{attribute 'reflection'}
FUNCTION_BLOCK FB_RS485_EASTRON_SDM630_MQTT EXTENDS FB_MQTT_BASE IMPLEMENTS I_RS485_DEVICE
  VAR
    {attribute 'noinit'}
    {attribute 'instance-path'}
    sInstancePath : STRING(GVL_MQTT.MQTT_TOPIC_LEN);  (* object's full instance name *)
    bIsDataUpdated : BOOL := FALSE;
    fbTimerData : TON;
    stStep : ST_RS485_STEP;  (* One read covers the whole measurement block: function 4 (input registers), 64 words from 16#000C (phase 1 power) to 16#004B (total export energy). Reading it in one stStep keeps the values consistent with each other and costs the bus one slot instead of 26. Filled by FB_init in code rather than by a declaration initialiser, which a script cannot revise once the compiler has stored it. *)
    fbMqttDiscoveryDevice : FB_EASTRON_SDM_MQTT_DISCOVERY_DEVICE;  (* Owned rather than referenced, unlike the 1-Wire sensors which share a gateway device from the GVL: a meter is one Home Assistant device on its own, so there is nothing to share and self-wiring has nothing to look up. *)
  END_VAR
  VAR_OUTPUT
    L1_ACTIVEPOWER : REAL := 0;
    L2_ACTIVEPOWER : REAL := 0;  (* L1 Active Power. SDM630 input register 16#000C. *)
    L3_ACTIVEPOWER : REAL := 0;  (* L2 Active Power. SDM630 input register 16#000E. *)
    L1_VA : REAL := 0;  (* L3 Active Power. SDM630 input register 16#0010. *)
    L2_VA : REAL := 0;  (* L1 Apparent Power. SDM630 input register 16#0012. *)
    L3_VA : REAL := 0;  (* L2 Apparent Power. SDM630 input register 16#0014. *)
    L1_VAR : REAL := 0;  (* L3 Apparent Power. SDM630 input register 16#0016. *)
    L2_VAR : REAL := 0;  (* L1 Reactive Power. SDM630 input register 16#0018. *)
    L3_VAR : REAL := 0;  (* L2 Reactive Power. SDM630 input register 16#001A. *)
    L1_PF : REAL := 0;  (* L3 Reactive Power. SDM630 input register 16#001C. *)
    L2_PF : REAL := 0;  (* L1 Power Factor. SDM630 input register 16#001E. *)
    L3_PF : REAL := 0;  (* L2 Power Factor. SDM630 input register 16#0020. *)
    L1_PHI : REAL := 0;  (* L3 Power Factor. SDM630 input register 16#0022. *)
    L2_PHI : REAL := 0;  (* L1 Phase Angle. SDM630 input register 16#0024. *)
    L3_PHI : REAL := 0;  (* L2 Phase Angle. SDM630 input register 16#0026. *)
    AVG_LN_V : REAL := 0;  (* L3 Phase Angle. SDM630 input register 16#0028. *)
    AVG_LINE_I : REAL := 0;  (* Average L-iN Voltage. SDM630 input register 16#002A. *)
    SUM_LINE_I : REAL := 0;  (* Average Line Current. SDM630 input register 16#002C. *)
    ACTIVEPOWER : REAL := 0;  (* Sum of Line Currents. SDM630 input register 16#002E. *)
    TOTAL_VA : REAL := 0;  (* Active Power. SDM630 input register 16#0034. *)
    TOTAL_VAR : REAL := 0;  (* Total Apparent Power. SDM630 input register 16#0038. *)
    TOTAL_PF : REAL := 0;  (* Total Reactive Power. SDM630 input register 16#003C. *)
    TOTAL_PHI : REAL := 0;  (* Total Power Factor. SDM630 input register 16#003E. *)
    FREQUENCY : REAL := 0;  (* Total Phase Angle. SDM630 input register 16#0042. *)
    TOTAL_IMPORT_ENERGY : REAL := 0;  (* Frequency. SDM630 input register 16#0046. *)
    TOTAL_EXPORT_ENERGY : REAL := 0;  (* Total Import Energy. SDM630 input register 16#0048. *)
    DataAvailable : BOOL := FALSE;  (* Total Export Energy. SDM630 input register 16#004A. *)
    Error : BOOL := FALSE;
  END_VAR

            (* --- self-wiring prologue ----------------------------------------------------
   Makes the InitMqtt and InitMqttDiscovery calls optional. Set FriendlyName at
   the declaration site and this block wires itself from GVL_MQTT on its
   first cyclic call, then announces itself to Home Assistant.

   Deliberately in the body rather than in FB_init: it dereferences GVL members
   and reads the reflection instance path, and doing that during initialisation
   would rely on an ordering nothing enforces and the compiler cannot check. The
   body is the same lifecycle phase the init actions used, so this is not merely
   safe, it is the phase that already works today.

   The wiring calls this block's own unmodified InitMqtt / InitMqttDiscovery
   methods, so anything published - topics and discovery JSON alike - is produced
   by exactly the code that produces it today. Only the trigger moved.

   Dormant while FriendlyName is empty, so existing projects and existing call
   sites keep working untouched.

   A block wired this way MUST be called cyclically. An instance whose body never
   runs is now unwired and absent from Home Assistant, where the init action used
   to wire it regardless. Nothing warns about that.  *)
IF FriendlyName <> '' THEN

	IF NOT bInitMqttDone THEN
		THIS^.InitMqtt(
			MQTTPublishPrefix := ADR(GVL_MQTT.MqttPubRS485Prefix),
			pMqttPublishQueue := ADR(GVL_MQTT.fbMqttPublishQueue));
	END_IF

	IF bInitMqttDone AND NOT bInitMqttDiscoveryDone THEN
		THIS^.InitMqttDiscovery(
			Device := ADR(THIS^.fbMqttDiscoveryDevice),
			DeviceName := FriendlyName);
	END_IF

END_IF

fbTimerData();

(* Publish on change of data rather than on a timer: ProcessDataArray sets the
   flag when a response arrives, so the publish rate follows DataPollingInterval
   and nothing is republished while the bus is quiet. PubMqttMessage is a no-op
   until InitMqtt has run, so this needs no further guard. *)
IF bIsDataUpdated THEN
	bIsDataUpdated := FALSE;

	PubMqttMessage(Suffix := '/L1_ACTP', Data := REAL_TO_STRING(L1_ACTIVEPOWER));
	PubMqttMessage(Suffix := '/L2_ACTP', Data := REAL_TO_STRING(L2_ACTIVEPOWER));
	PubMqttMessage(Suffix := '/L3_ACTP', Data := REAL_TO_STRING(L3_ACTIVEPOWER));
	PubMqttMessage(Suffix := '/L1_VA', Data := REAL_TO_STRING(L1_VA));
	PubMqttMessage(Suffix := '/L2_VA', Data := REAL_TO_STRING(L2_VA));
	PubMqttMessage(Suffix := '/L3_VA', Data := REAL_TO_STRING(L3_VA));
	PubMqttMessage(Suffix := '/L1_VAR', Data := REAL_TO_STRING(L1_VAR));
	PubMqttMessage(Suffix := '/L2_VAR', Data := REAL_TO_STRING(L2_VAR));
	PubMqttMessage(Suffix := '/L3_VAR', Data := REAL_TO_STRING(L3_VAR));
	PubMqttMessage(Suffix := '/L1_PF', Data := REAL_TO_STRING(L1_PF));
	PubMqttMessage(Suffix := '/L2_PF', Data := REAL_TO_STRING(L2_PF));
	PubMqttMessage(Suffix := '/L3_PF', Data := REAL_TO_STRING(L3_PF));
	PubMqttMessage(Suffix := '/L1_PHI', Data := REAL_TO_STRING(L1_PHI));
	PubMqttMessage(Suffix := '/L2_PHI', Data := REAL_TO_STRING(L2_PHI));
	PubMqttMessage(Suffix := '/L3_PHI', Data := REAL_TO_STRING(L3_PHI));
	PubMqttMessage(Suffix := '/AVG_V', Data := REAL_TO_STRING(AVG_LN_V));
	PubMqttMessage(Suffix := '/AVG_I', Data := REAL_TO_STRING(AVG_LINE_I));
	PubMqttMessage(Suffix := '/SUM_I', Data := REAL_TO_STRING(SUM_LINE_I));
	PubMqttMessage(Suffix := '/ACTP', Data := REAL_TO_STRING(ACTIVEPOWER));
	PubMqttMessage(Suffix := '/TOT_VA', Data := REAL_TO_STRING(TOTAL_VA));
	PubMqttMessage(Suffix := '/TOT_VAR', Data := REAL_TO_STRING(TOTAL_VAR));
	PubMqttMessage(Suffix := '/TOT_PF', Data := REAL_TO_STRING(TOTAL_PF));
	PubMqttMessage(Suffix := '/TOT_PHI', Data := REAL_TO_STRING(TOTAL_PHI));
	PubMqttMessage(Suffix := '/FREQ', Data := REAL_TO_STRING(FREQUENCY));
	PubMqttMessage(Suffix := '/IMPE', Data := REAL_TO_STRING(TOTAL_IMPORT_ENERGY));
	PubMqttMessage(Suffix := '/EXPE', Data := REAL_TO_STRING(TOTAL_EXPORT_ENERGY));
END_IF
          

METHOD HasWork : E_RS485_WORK_LEVEL
                  IF fbTimerData.Q THEN
	HasWork := E_RS485_WORK_LEVEL.POLL;
ELSE
	HasWork := E_RS485_WORK_LEVEL.NONE;
END_IF

                
END_METHOD

METHOD OnStepResult
  VAR_INPUT
    StepIndex : INT;
    Failed : BOOL;
    pData : POINTER TO A_RS485_READ_BUFFER;
    Count : INT;
  END_VAR
                  THIS^.Error := Failed;
THIS^.fbTimerData.IN := TRUE;

IF NOT Failed AND Count >= 64 THEN
	(* Every value is a big-endian IEEE float across two consecutive words, so the
	   word index is the register offset from 16#000C doubled. Gaps below are
	   registers the SDM630 reserves. *)
	THIS^.L1_ACTIVEPOWER := F_SWAP_WORDS_TO_REAL(pData^[0], pData^[1]);	// 16#000C L1 Active Power
	THIS^.L2_ACTIVEPOWER := F_SWAP_WORDS_TO_REAL(pData^[2], pData^[3]);	// 16#000E L2 Active Power
	THIS^.L3_ACTIVEPOWER := F_SWAP_WORDS_TO_REAL(pData^[4], pData^[5]);	// 16#0010 L3 Active Power
	THIS^.L1_VA := F_SWAP_WORDS_TO_REAL(pData^[6], pData^[7]);	// 16#0012 L1 Apparent Power
	THIS^.L2_VA := F_SWAP_WORDS_TO_REAL(pData^[8], pData^[9]);	// 16#0014 L2 Apparent Power
	THIS^.L3_VA := F_SWAP_WORDS_TO_REAL(pData^[10], pData^[11]);	// 16#0016 L3 Apparent Power
	THIS^.L1_VAR := F_SWAP_WORDS_TO_REAL(pData^[12], pData^[13]);	// 16#0018 L1 Reactive Power
	THIS^.L2_VAR := F_SWAP_WORDS_TO_REAL(pData^[14], pData^[15]);	// 16#001A L2 Reactive Power
	THIS^.L3_VAR := F_SWAP_WORDS_TO_REAL(pData^[16], pData^[17]);	// 16#001C L3 Reactive Power
	THIS^.L1_PF := F_SWAP_WORDS_TO_REAL(pData^[18], pData^[19]);	// 16#001E L1 Power Factor
	THIS^.L2_PF := F_SWAP_WORDS_TO_REAL(pData^[20], pData^[21]);	// 16#0020 L2 Power Factor
	THIS^.L3_PF := F_SWAP_WORDS_TO_REAL(pData^[22], pData^[23]);	// 16#0022 L3 Power Factor
	THIS^.L1_PHI := F_SWAP_WORDS_TO_REAL(pData^[24], pData^[25]);	// 16#0024 L1 Phase Angle
	THIS^.L2_PHI := F_SWAP_WORDS_TO_REAL(pData^[26], pData^[27]);	// 16#0026 L2 Phase Angle
	THIS^.L3_PHI := F_SWAP_WORDS_TO_REAL(pData^[28], pData^[29]);	// 16#0028 L3 Phase Angle
	THIS^.AVG_LN_V := F_SWAP_WORDS_TO_REAL(pData^[30], pData^[31]);	// 16#002A Average L-iN Voltage
	THIS^.AVG_LINE_I := F_SWAP_WORDS_TO_REAL(pData^[32], pData^[33]);	// 16#002C Average Line Current
	THIS^.SUM_LINE_I := F_SWAP_WORDS_TO_REAL(pData^[34], pData^[35]);	// 16#002E Sum of Line Currents
	THIS^.ACTIVEPOWER := F_SWAP_WORDS_TO_REAL(pData^[40], pData^[41]);	// 16#0034 Active Power
	THIS^.TOTAL_VA := F_SWAP_WORDS_TO_REAL(pData^[44], pData^[45]);	// 16#0038 Total Apparent Power
	THIS^.TOTAL_VAR := F_SWAP_WORDS_TO_REAL(pData^[48], pData^[49]);	// 16#003C Total Reactive Power
	THIS^.TOTAL_PF := F_SWAP_WORDS_TO_REAL(pData^[50], pData^[51]);	// 16#003E Total Power Factor
	THIS^.TOTAL_PHI := F_SWAP_WORDS_TO_REAL(pData^[54], pData^[55]);	// 16#0042 Total Phase Angle
	THIS^.FREQUENCY := F_SWAP_WORDS_TO_REAL(pData^[58], pData^[59]);	// 16#0046 Frequency
	THIS^.TOTAL_IMPORT_ENERGY := F_SWAP_WORDS_TO_REAL(pData^[60], pData^[61]);	// 16#0048 Total Import Energy
	THIS^.TOTAL_EXPORT_ENERGY := F_SWAP_WORDS_TO_REAL(pData^[62], pData^[63]);	// 16#004A Total Export Energy

	THIS^.DataAvailable := TRUE;
	THIS^.bIsDataUpdated := TRUE;
END_IF

                
END_METHOD

METHOD BuildTransaction : INT
  VAR_INPUT
    pSteps : POINTER TO A_RS485_STEP_LIST;
  END_VAR
  VAR
    iN : INT;
  END_VAR
                  IF fbTimerData.Q THEN
	pSteps^[0]			:= stStep;
	fbTimerData.IN		:= FALSE;
	BuildTransaction	:= 1;
ELSE
	BuildTransaction := 0;
END_IF

                
END_METHOD

METHOD InitMqttDiscovery
  VAR_INPUT
    Device : POINTER TO FB_EASTRON_SDM_MQTT_DISCOVERY_DEVICE;
    DeviceName : STRING(50);
    Model : STRING(20) := 'SDM630';
    overruleId : STRING(255) := '';
  END_VAR
  VAR
    id : STRING(255);
  END_VAR
                  (* Announces the meter as a device of its own, then one sensor entity per
   measurement. StateClass is what puts the two kWh totals into the Home
   Assistant energy dashboard; the instantaneous values are 'measurement' and
   power factor, phase angle, voltage, current and frequency carry none. *)
IF bInitMqttDone AND NOT bInitMqttDiscoveryDone THEN

	id := SUPER^.ResolveEntityId(overruleId := overruleId);

	Device^.initEastronDevice(
		name := DeviceName,
		id := id,
		Model := Model,
		availabilityTopic1 := GVL_MQTT.MqttAvailabilityTopic,
		availabilityTopic2 := CONCAT(THIS^.sMQTTPublishTopic, '/availability'),
		availabilityOnline := GVL_MQTT.MqttAvailabilityOnlinePayload,
		availabilityOffline := GVL_MQTT.MqttAvailabilityOfflinePayload,
		MqttDiscoveryPrefix := GVL_MQTT.MqttHADiscoveryPrefix,
		MqttDiagnosticTopic := CONCAT(THIS^.sMQTTPublishTopic, '/diagnostic'),
		pMqttPublishQueue := ADR(GVL_MQTT.fbMqttPublishQueue));

(* This device publishes from the RS485 task, so its messages take that
   task's queue lane. A lane may only ever have one producing task. *)
Device^.SetLane(Lane := GVL_MQTT.MQTT_LANE_RS485);

	Device^.CreateSensorEntity(
		Name := 'L1 Active Power',
		Id := CONCAT(id, '_L1_ACTP'),
		StateTopic := CONCAT(THIS^.sMQTTPublishTopic, '/L1_ACTP'),
		DeviceClass := 'power',
		StateClass := 'measurement',
		UnitOfMeasurement := 'W');

	Device^.CreateSensorEntity(
		Name := 'L2 Active Power',
		Id := CONCAT(id, '_L2_ACTP'),
		StateTopic := CONCAT(THIS^.sMQTTPublishTopic, '/L2_ACTP'),
		DeviceClass := 'power',
		StateClass := 'measurement',
		UnitOfMeasurement := 'W');

	Device^.CreateSensorEntity(
		Name := 'L3 Active Power',
		Id := CONCAT(id, '_L3_ACTP'),
		StateTopic := CONCAT(THIS^.sMQTTPublishTopic, '/L3_ACTP'),
		DeviceClass := 'power',
		StateClass := 'measurement',
		UnitOfMeasurement := 'W');

	Device^.CreateSensorEntity(
		Name := 'L1 Apparent Power',
		Id := CONCAT(id, '_L1_VA'),
		StateTopic := CONCAT(THIS^.sMQTTPublishTopic, '/L1_VA'),
		DeviceClass := 'apparent_power',
		StateClass := 'measurement',
		UnitOfMeasurement := 'VA');

	Device^.CreateSensorEntity(
		Name := 'L2 Apparent Power',
		Id := CONCAT(id, '_L2_VA'),
		StateTopic := CONCAT(THIS^.sMQTTPublishTopic, '/L2_VA'),
		DeviceClass := 'apparent_power',
		StateClass := 'measurement',
		UnitOfMeasurement := 'VA');

	Device^.CreateSensorEntity(
		Name := 'L3 Apparent Power',
		Id := CONCAT(id, '_L3_VA'),
		StateTopic := CONCAT(THIS^.sMQTTPublishTopic, '/L3_VA'),
		DeviceClass := 'apparent_power',
		StateClass := 'measurement',
		UnitOfMeasurement := 'VA');

	Device^.CreateSensorEntity(
		Name := 'L1 Reactive Power',
		Id := CONCAT(id, '_L1_VAR'),
		StateTopic := CONCAT(THIS^.sMQTTPublishTopic, '/L1_VAR'),
		DeviceClass := 'reactive_power',
		StateClass := 'measurement',
		UnitOfMeasurement := 'var');

	Device^.CreateSensorEntity(
		Name := 'L2 Reactive Power',
		Id := CONCAT(id, '_L2_VAR'),
		StateTopic := CONCAT(THIS^.sMQTTPublishTopic, '/L2_VAR'),
		DeviceClass := 'reactive_power',
		StateClass := 'measurement',
		UnitOfMeasurement := 'var');

	Device^.CreateSensorEntity(
		Name := 'L3 Reactive Power',
		Id := CONCAT(id, '_L3_VAR'),
		StateTopic := CONCAT(THIS^.sMQTTPublishTopic, '/L3_VAR'),
		DeviceClass := 'reactive_power',
		StateClass := 'measurement',
		UnitOfMeasurement := 'var');

	Device^.CreateSensorEntity(
		Name := 'L1 Power Factor',
		Id := CONCAT(id, '_L1_PF'),
		StateTopic := CONCAT(THIS^.sMQTTPublishTopic, '/L1_PF'),
		DeviceClass := 'power_factor',
		UnitOfMeasurement := '');

	Device^.CreateSensorEntity(
		Name := 'L2 Power Factor',
		Id := CONCAT(id, '_L2_PF'),
		StateTopic := CONCAT(THIS^.sMQTTPublishTopic, '/L2_PF'),
		DeviceClass := 'power_factor',
		UnitOfMeasurement := '');

	Device^.CreateSensorEntity(
		Name := 'L3 Power Factor',
		Id := CONCAT(id, '_L3_PF'),
		StateTopic := CONCAT(THIS^.sMQTTPublishTopic, '/L3_PF'),
		DeviceClass := 'power_factor',
		UnitOfMeasurement := '');

	Device^.CreateSensorEntity(
		Name := 'L1 Phase Angle',
		Id := CONCAT(id, '_L1_PHI'),
		StateTopic := CONCAT(THIS^.sMQTTPublishTopic, '/L1_PHI'),
		DeviceClass := '',
		UnitOfMeasurement := '°');

	Device^.CreateSensorEntity(
		Name := 'L2 Phase Angle',
		Id := CONCAT(id, '_L2_PHI'),
		StateTopic := CONCAT(THIS^.sMQTTPublishTopic, '/L2_PHI'),
		DeviceClass := '',
		UnitOfMeasurement := '°');

	Device^.CreateSensorEntity(
		Name := 'L3 Phase Angle',
		Id := CONCAT(id, '_L3_PHI'),
		StateTopic := CONCAT(THIS^.sMQTTPublishTopic, '/L3_PHI'),
		DeviceClass := '',
		UnitOfMeasurement := '°');

	Device^.CreateSensorEntity(
		Name := 'Average L-N Voltage',
		Id := CONCAT(id, '_AVG_V'),
		StateTopic := CONCAT(THIS^.sMQTTPublishTopic, '/AVG_V'),
		DeviceClass := 'voltage',
		UnitOfMeasurement := 'V');

	Device^.CreateSensorEntity(
		Name := 'Average Line Current',
		Id := CONCAT(id, '_AVG_I'),
		StateTopic := CONCAT(THIS^.sMQTTPublishTopic, '/AVG_I'),
		DeviceClass := 'current',
		UnitOfMeasurement := 'A');

	Device^.CreateSensorEntity(
		Name := 'Sum of Line Currents',
		Id := CONCAT(id, '_SUM_I'),
		StateTopic := CONCAT(THIS^.sMQTTPublishTopic, '/SUM_I'),
		DeviceClass := 'current',
		UnitOfMeasurement := 'A');

	Device^.CreateSensorEntity(
		Name := 'Active Power',
		Id := CONCAT(id, '_ACTP'),
		StateTopic := CONCAT(THIS^.sMQTTPublishTopic, '/ACTP'),
		DeviceClass := 'power',
		StateClass := 'measurement',
		UnitOfMeasurement := 'W');

	Device^.CreateSensorEntity(
		Name := 'Total Apparent Power',
		Id := CONCAT(id, '_TOT_VA'),
		StateTopic := CONCAT(THIS^.sMQTTPublishTopic, '/TOT_VA'),
		DeviceClass := 'apparent_power',
		StateClass := 'measurement',
		UnitOfMeasurement := 'VA');

	Device^.CreateSensorEntity(
		Name := 'Total Reactive Power',
		Id := CONCAT(id, '_TOT_VAR'),
		StateTopic := CONCAT(THIS^.sMQTTPublishTopic, '/TOT_VAR'),
		DeviceClass := 'reactive_power',
		StateClass := 'measurement',
		UnitOfMeasurement := 'var');

	Device^.CreateSensorEntity(
		Name := 'Total Power Factor',
		Id := CONCAT(id, '_TOT_PF'),
		StateTopic := CONCAT(THIS^.sMQTTPublishTopic, '/TOT_PF'),
		DeviceClass := 'power_factor',
		UnitOfMeasurement := '');

	Device^.CreateSensorEntity(
		Name := 'Total Phase Angle',
		Id := CONCAT(id, '_TOT_PHI'),
		StateTopic := CONCAT(THIS^.sMQTTPublishTopic, '/TOT_PHI'),
		DeviceClass := '',
		UnitOfMeasurement := '°');

	Device^.CreateSensorEntity(
		Name := 'Frequency',
		Id := CONCAT(id, '_FREQ'),
		StateTopic := CONCAT(THIS^.sMQTTPublishTopic, '/FREQ'),
		DeviceClass := 'frequency',
		UnitOfMeasurement := 'Hz');

	Device^.CreateSensorEntity(
		Name := 'Total Import Energy',
		Id := CONCAT(id, '_IMP_ENERG'),
		StateTopic := CONCAT(THIS^.sMQTTPublishTopic, '/IMPE'),
		DeviceClass := 'energy',
		StateClass := 'total_increasing',
		UnitOfMeasurement := 'kWh');

	Device^.CreateSensorEntity(
		Name := 'Total Export Energy',
		Id := CONCAT(id, '_EXP_ENERG'),
		StateTopic := CONCAT(THIS^.sMQTTPublishTopic, '/EXPE'),
		DeviceClass := 'energy',
		StateClass := 'total_increasing',
		UnitOfMeasurement := 'kWh');

	bInitMqttDiscoveryDone := TRUE;
END_IF
                
END_METHOD

METHOD PubMqttMessage
  VAR_INPUT
    Suffix : STRING(100);
    Data : STRING(100);
  END_VAR
                  IF bInitMqttDone THEN
		pMqttPublishQueue^.AddMessageOn(Lane := GVL_MQTT.MQTT_LANE_RS485,
			Payload := Data,
			Topic := CONCAT(THIS^.sMQTTPublishTopic, Suffix),
			Qos := MQTT.QoS.ExactlyOnce,
			MqttRetain := FALSE
		);
END_IF
                
END_METHOD

METHOD InitMqtt
  VAR_INPUT
    MQTTPublishPrefix : POINTER TO STRING;
    pMqttPublishQueue : POINTER TO FB_MQTT_PUBLISH_QUEUE;
  END_VAR
                  SUPER^._sInstancePath := THIS^.sInstancePath; // Due to reflection its location is important

(*pass trough*)
THIS^.pMqttPublishQueue := pMqttPublishQueue;
THIS^.psMqttPublishTopicPrefix := MQTTPublishPrefix;

SUPER^.InitBaseMqtt();
                
END_METHOD

METHOD FB_init : BOOL
  VAR_INPUT
    bInitRetains : BOOL;  (* TRUE: the retain variables are initialized (reset warm / reset cold) *)
    bInCopyCode : BOOL;  (* TRUE: the instance will be copied to the copy code afterward (online change) *)
    DeviceAddress : BYTE;  (* Modbus slave address of the meter. *)
    DataPollingInterval : TIME;  (* How often the meter is read. One read covers all 26 measurements. *)
  END_VAR
                  (* Modbus address and poll rate describe the wiring, not a mode, so they are
   fixed for the life of the instance and belong here rather than in a runtime
   setter. Note the consequence: changing either afterwards means editing the
   declaration in the IDE - CODESYS stores an instance's FB_init arguments beside
   the declaration text, where no script can reach them. *)
THIS^.stStep.DeviceId		:= DeviceAddress;
THIS^.stStep.FunctionCode	:= 4;
THIS^.stStep.Address		:= 12;	(* 16#000C, phase 1 active power *)
THIS^.stStep.Quantity		:= 64;	(* through 16#004B, total export energy *)

THIS^.fbTimerData.PT := DataPollingInterval;
THIS^.fbTimerData.IN := TRUE;

FB_init := TRUE;

                
END_METHOD

METHOD OnTransactionDone
  VAR_INPUT
    StepsRun : INT;
    Failures : INT;
  END_VAR
                  (* One announcement per transaction, at the point the bus is released. *)
IF StepsRun > 0 AND Failures >= StepsRun THEN
	PubMqttMessage(Suffix := '/availability', Data := 'offline');
ELSIF StepsRun > 0 THEN
	PubMqttMessage(Suffix := '/availability', Data := 'online');
END_IF

                
END_METHOD

(* Nothing to commission on this device. See I_RS485_DEVICE.GetCommissioning. *)
METHOD GetCommissioning : BOOL
  VAR_INPUT
    BusBaudrate : UDINT;
    pRequest : POINTER TO ST_RS485_COMMISSION_REQUEST;
  END_VAR
                  (* Nothing to commission. This device is configured on the device itself - switches,
   a display, or a factory setting that already matches this bus - so it answers at
   whatever the bus runs at and there is nothing for the commissioner to write.

   Which is the ordinary case: the cost of the whole mechanism, for a device like
   this one, is this method call once at startup. *)
GetCommissioning := FALSE;

                
END_METHOD
END_FUNCTION_BLOCK

{attribute 'reflection'}
FUNCTION_BLOCK FB_RS485_ESERA_OWD_MQTT EXTENDS FB_MQTT_BASE IMPLEMENTS I_RS485_DEVICE
  VAR
    {attribute 'noinit'}
    {attribute 'instance-path'}
    sInstancePath : STRING(GVL_MQTT.MQTT_TOPIC_LEN);  (* object's full instance name *)
    OwdNumber : UINT;
    fbTimerData : TON;
    stStep : ST_RS485_STEP;  (* One read of the gateway's per-sensor block: function 3, 17 holding registers from OwdNumber * 100. Filled by FB_init in code. *)
    pMqttDiscoveryDevice : POINTER TO FB_1WIRE_MQTT_DISCOVERY_DEVICE;
    uiAllowedErrorCount : UINT := 3;
    uiCurrentErrorCount : UINT := 0;
  END_VAR
  VAR_OUTPUT
    OWD_VOLTAGE : REAL := 0;
    TEMPERATURE : REAL := 0;
    HUMIDITY : REAL := 0;
    DEW_POINT : REAL := 0;
    AIR_QUALITY : REAL := 0;
    BRIGHTNESS : REAL := 0;
    DataAvailable : BOOL := FALSE;
    Error : BOOL := FALSE;
  END_VAR

            fbTimerData();


          

METHOD HasWork : E_RS485_WORK_LEVEL
                  IF fbTimerData.Q THEN
	HasWork := E_RS485_WORK_LEVEL.POLL;
ELSE
	HasWork := E_RS485_WORK_LEVEL.NONE;
END_IF

                
END_METHOD

METHOD OnStepResult
  VAR_INPUT
    StepIndex : INT;
    Failed : BOOL;
    pData : POINTER TO A_RS485_READ_BUFFER;
    Count : INT;
  END_VAR
                  THIS^.fbTimerData.IN := TRUE;

(* Register 12 is the gateway's own status word for this sensor: non-zero means
   the gateway answered but the 1-Wire device behind it did not. A short reply
   is treated the same way - there is no status to trust. *)
IF Failed OR Count < 17 OR WORD_TO_INT(pData^[12]) <> 0 THEN
	THIS^.Error := TRUE;
	(* A single miss is normal on a 1-Wire bus, so availability only drops after
	   uiAllowedErrorCount of them in a row. *)
	IF THIS^.uiCurrentErrorCount >= THIS^.uiAllowedErrorCount THEN
		PubMqttMessage(Suffix := '/availability', Data := 'offline');
	END_IF
	THIS^.uiCurrentErrorCount := THIS^.uiCurrentErrorCount + 1;
	RETURN;
END_IF

THIS^.Error := FALSE;
THIS^.DataAvailable := TRUE;
THIS^.uiCurrentErrorCount := 0;
PubMqttMessage(Suffix := '/availability', Data := 'online');

IF bInitMqttDiscoveryDone THEN
	THIS^.pMqttDiscoveryDevice^.SendDeviceUpdate(Model := WORD_TO_STRING(pData^[16]));
END_IF

// Data handling
IF pData^[16] = 11151 OR pData^[16] = 11152 THEN // Temperature, humidity & air quality
	ProcessTemperature(pData^[0]);
	ProcessOwdVoltage(pData^[2]);
	ProcessHumidity(pData^[4]);
	ProcessDewPoint(pData^[6]);
	ProcessAirQuality(pData^[8]);
ELSIF pData^[16] = 11102 OR pData^[16] = 11113 OR pData^[16] = 11120 OR pData^[16] = 11148 OR pData^[16] = 11150 OR pData^[16] = 11160 THEN // Temperature, humidity
	ProcessTemperature(pData^[0]);
	ProcessOwdVoltage(pData^[2]);
	ProcessHumidity(pData^[4]);
	ProcessDewPoint(pData^[6]);
ELSIF pData^[16] = 11121 OR pData^[16] = 11132 OR pData^[16] = 11134 OR pData^[16] = 11135 THEN // Temperature, humidity, brightness
	ProcessTemperature(pData^[0]);
	ProcessOwdVoltage(pData^[2]);
	ProcessHumidity(pData^[4]);
	ProcessDewPoint(pData^[6]);
	ProcessBrigthness(pData^[8]);
ELSIF pData^[16] = 1820 THEN // Temperature DS18B20
	ProcessTemperature(pData^[0]);
END_IF

                
END_METHOD

METHOD BuildTransaction : INT
  VAR_INPUT
    pSteps : POINTER TO A_RS485_STEP_LIST;
  END_VAR
  VAR
    iN : INT;
  END_VAR
                  IF fbTimerData.Q THEN
	pSteps^[0]			:= stStep;
	fbTimerData.IN		:= FALSE;
	BuildTransaction	:= 1;
ELSE
	BuildTransaction := 0;
END_IF

                
END_METHOD

METHOD InitMqttDiscovery
  VAR_INPUT
    Device : POINTER TO FB_1WIRE_MQTT_DISCOVERY_DEVICE;
    ParentDevice : POINTER TO FB_PLC_MQTT_DISCOVERY_DEVICE;
    DeviceName : STRING(50);
    SupportsTemperature : BOOL := FALSE;
    SupportsHumidity : BOOL := FALSE;
    SupportsCO2 : BOOL := FALSE;
    SupportsDewPoint : BOOL := FALSE;
    SupportsBrightness : BOOL := FALSE;
    SupportsOwdVoltage : BOOL := FALSE;
  END_VAR
  VAR
    id : STRING(255);
  END_VAR
                  IF bInitMqttDone AND NOT bInitMqttDiscoveryDone THEN
	
	THIS^.pMqttDiscoveryDevice := Device;
	
	id := SUPER^.ResolveEntityId(overruleId := '');
	
	Device^.init1WireDevice(
		name := DeviceName,
		id := id,
		deviceAvailabilityTopic := CONCAT(THIS^.sMQTTPublishTopic, '/availability'),
		deviceDiagnosticTopic := CONCAT(THIS^.sMQTTPublishTopic, '/diagnostic'));

(* This device publishes from the RS485 task, so its messages take that
   task's queue lane. A lane may only ever have one producing task. *)
Device^.SetLane(Lane := GVL_MQTT.MQTT_LANE_RS485);
		
	IF SupportsTemperature THEN
		Device^.CreateSensorEntity(
			Name := 'Temperature',
			Id := CONCAT(id, '_TEMP'),
			StateTopic := CONCAT(THIS^.sMQTTPublishTopic, '/TEMP'),
			DeviceClass := 'temperature',
			UnitOfMeasurement := '°C'); 
	END_IF;	
	
	IF SupportsHumidity THEN
		Device^.CreateSensorEntity(
			Name := 'Humidity',
			Id := CONCAT(id, '_HUM'),
			StateTopic := CONCAT(THIS^.sMQTTPublishTopic, '/HUM'),
			DeviceClass := 'humidity',
			UnitOfMeasurement := '%');
	END_IF;
	
	IF SupportsCO2 THEN
		Device^.CreateSensorEntity(
			Name := 'Carbon Dioxide',
			Id := CONCAT(id, '_CO2'),
			StateTopic := CONCAT(THIS^.sMQTTPublishTopic, '/CO2'),
			DeviceClass := 'carbon_dioxide',
			UnitOfMeasurement := 'ppm');
	END_IF;
	
	IF SupportsDewPoint THEN
		Device^.CreateSensorEntity(
			Name := 'Dew Point',
			Id := CONCAT(id, '_DEWP'),
			StateTopic := CONCAT(THIS^.sMQTTPublishTopic, '/DEWP'),
			DeviceClass := 'temperature',
			UnitOfMeasurement := '°C'); 
	END_IF;	
	
	IF SupportsBrightness THEN
		Device^.CreateSensorEntity(
			Name := 'Brightness',
			Id := CONCAT(id, '_ILLUM'),
			StateTopic := CONCAT(THIS^.sMQTTPublishTopic, '/ILLUM'),
			DeviceClass := 'illuminance');
	END_IF;	
	
	IF SupportsOwdVoltage THEN
		Device^.CreateDiagnosticSensorEntity(
			Name := 'Operating Voltage',
			Id := CONCAT(id, '_OWDV'),
			StateTopic := CONCAT(THIS^.sMQTTPublishTopic, '/OWDV'));
	END_IF;

	bInitMqttDiscoveryDone := TRUE;
END_IF
                
END_METHOD

METHOD InitMqtt
  VAR_INPUT
    MQTTPublishPrefix : POINTER TO STRING;
    pMqttPublishQueue : POINTER TO FB_MQTT_PUBLISH_QUEUE;
  END_VAR
                  SUPER^._sInstancePath := THIS^.sInstancePath; // Due to reflection its location is important

(*pass trough*)
THIS^.pMqttPublishQueue := pMqttPublishQueue;
THIS^.psMqttPublishTopicPrefix:=MQTTPublishPrefix;
SUPER^.InitBaseMqtt();

                
END_METHOD

METHOD PubMqttMessage
  VAR_INPUT
    Suffix : STRING(100);
    Data : STRING(100);
  END_VAR
                  IF bInitMqttDone THEN
		pMqttPublishQueue^.AddMessageOn(Lane := GVL_MQTT.MQTT_LANE_RS485,
			Payload := Data,
			Topic := CONCAT(CONCAT(psMqttPublishTopicPrefix^, MqttPublishTopicSuffix), Suffix),
			Qos := MQTT.QoS.ExactlyOnce,
			MqttRetain := FALSE
		);
END_IF
                
END_METHOD

METHOD ProcessTemperature
  VAR_INPUT
    Data : WORD;
  END_VAR
                  (* Signed: the gateway scales by 100 and encodes two's complement, and both
   of these read below zero on an outdoor sensor. Unsigned turned -1 degree
   into +655.35 and nothing could report frost. *)
THIS^.TEMPERATURE := INT_TO_REAL(WORD_TO_INT(Data)) / 100;
PubMqttMessage(Suffix := '/TEMP', Data := REAL_TO_STRING(TEMPERATURE));
                
END_METHOD

METHOD ProcessOwdVoltage
  VAR_INPUT
    Data : WORD;
  END_VAR
                  THIS^.OWD_VOLTAGE := WORD_TO_REAL(Data);
PubMqttMessage(Suffix := '/OWDV', Data := REAL_TO_STRING(OWD_VOLTAGE));
                
END_METHOD

METHOD ProcessHumidity
  VAR_INPUT
    Data : WORD;
  END_VAR
                  THIS^.HUMIDITY := WORD_TO_REAL(Data) / 100;
PubMqttMessage(Suffix := '/HUM', Data := REAL_TO_STRING(HUMIDITY));
                
END_METHOD

METHOD ProcessDewPoint
  VAR_INPUT
    Data : WORD;
  END_VAR
                  (* Signed: the gateway scales by 100 and encodes two's complement, and both
   of these read below zero on an outdoor sensor. Unsigned turned -1 degree
   into +655.35 and nothing could report frost. *)
THIS^.DEW_POINT := INT_TO_REAL(WORD_TO_INT(Data)) / 100;
PubMqttMessage(Suffix := '/DEWP', Data := REAL_TO_STRING(DEW_POINT));
                
END_METHOD

METHOD ProcessAirQuality
  VAR_INPUT
    Data : WORD;
  END_VAR
                  THIS^.AIR_QUALITY := WORD_TO_REAL(Data) / 100;
PubMqttMessage(Suffix := '/CO2', Data := REAL_TO_STRING(AIR_QUALITY));
                
END_METHOD

METHOD ProcessBrigthness
  VAR_INPUT
    Data : WORD;
  END_VAR
                  THIS^.BRIGHTNESS := WORD_TO_REAL(Data) / 100;
(* /ILLUM, matching the entity id and the StateTopic in InitMqttDiscovery.
   This published to /BNESS, so the illuminance entity never received a value. *)
PubMqttMessage(Suffix := '/ILLUM', Data := REAL_TO_STRING(BRIGHTNESS));
                
END_METHOD

(* FB_Init is always available implicitly and it is used primarily for initialization. The return value is not evaluated. For a specific influence, you can also declare the methods explicitly and provide additional code there with the standard initialization code. You can evaluate the return value. *)
METHOD FB_init : BOOL
  VAR_INPUT
    bInitRetains : BOOL;  (* TRUE: the retain variables are initialized (reset warm / reset cold) *)
    bInCopyCode : BOOL;  (* TRUE: the instance will be copied to the copy code afterward (online change) *)
    DeviceAddress : BYTE;
    OwdNumber : UINT;
    DataPollingInterval : TIME;
  END_VAR
                  THIS^.stStep.DeviceId		:= DeviceAddress;
THIS^.stStep.FunctionCode	:= 3;
THIS^.stStep.Address		:= OwdNumber * 100;
THIS^.stStep.Quantity		:= 17;

THIS^.fbTimerData.PT := DataPollingInterval;
THIS^.OwdNumber := OwdNumber;

THIS^.fbTimerData.IN := TRUE;

FB_Init := TRUE;

                
END_METHOD

METHOD OnTransactionDone
  VAR_INPUT
    StepsRun : INT;
    Failures : INT;
  END_VAR
                  (* Availability for this block is decided in OnStepResult, where the gateway's
   own status register and the consecutive-error count are both in scope. There
   is nothing left to announce here, and announcing it twice would undo the
   error tolerance. *)
;

                
END_METHOD

(* Nothing to commission on this device. See I_RS485_DEVICE.GetCommissioning. *)
METHOD GetCommissioning : BOOL
  VAR_INPUT
    BusBaudrate : UDINT;
    pRequest : POINTER TO ST_RS485_COMMISSION_REQUEST;
  END_VAR
                  (* Nothing to commission. This device is configured on the device itself - switches,
   a display, or a factory setting that already matches this bus - so it answers at
   whatever the bus runs at and there is nothing for the commissioner to write.

   Which is the ordinary case: the cost of the whole mechanism, for a device like
   this one, is this method call once at startup. *)
GetCommissioning := FALSE;

                
END_METHOD
END_FUNCTION_BLOCK

(* Modbus RTU master for the PFC's onboard serial port, behind I_RS485_TRANSPORT. This is the code that was proven on the bench in #182, lifted out of the RS485_RUN action into a block of its own and taught the write function codes it was missing. Two things about this hardware are baked in and deliberate: - Every reply arrives wrapped in glitch bytes - one 00 as the slave's driver enables, another as it releases, because the pair is undriven between frames. Measured across 34 consecutive captures: 34 leading nulls, 34 trailing nulls, 34 wCrc-bDataValid frames once trimmed. So the frame is trimmed and the wCrc judges what is left, rather than the iFirst byte being trusted. - The frame is delimited by silence, which is what RTU actually specifies, not by a byte count read out of the header. The counters are outputs on purpose. They are the only view of line quality this project has without a scope, and LeadNulls climbing in stStep with Ok is the normal healthy picture here, not a fault. *)
FUNCTION_BLOCK FB_RS485_TRANSPORT_RTU IMPLEMENTS I_RS485_TRANSPORT
  VAR_OUTPUT
    PortOpen : BOOL;  (* The serial port is open and usable *)
    PortError : BOOL;  (* SysComOpen2 failed; Reopen to try again *)
    Ok : UDINT;  (* Reply accepted *)
    CrcFail : UDINT;  (* Bytes arrived, wCrc over the trimmed frame was not zero *)
    NoReply : UDINT;  (* Nothing at all before the reply timeout *)
    ShortFrame : UDINT;  (* Too few bytes to be any bDataValid reply *)
    BadAddress : UDINT;  (* A well-formed frame from the wrong slave *)
    BadFunction : UDINT;  (* Right slave, function code we did not ask for *)
    BadEcho : UDINT;  (* Write acknowledged with the wrong address or value *)
    Exceptions : UDINT;  (* Slave answered with an exception reply *)
    LastException : BYTE;  (* Exception code from the most recent one *)
    LeadNulls : UDINT;  (* Not faults. On this hardware both should track Ok almost exactly. *)
    TrailNulls : UDINT;
    LastFailLen : UDINT;  (* The bytes of the most recent frame that would not check out, and how many there were. A counter can say a reply did not frame; only the bytes can say whether it was half a reply, two replies, an echo of the request, or noise - and those want different fixes. *)
    LastFailAddr : BYTE;
    LastFailFunc : BYTE;
    LastFailBytes : STRING(120);
  END_VAR
  VAR
    bConfigured : BOOL;  (* --- port ------------------------------------------------------------ *)
    stSettings : SysCom.SysComSettings;
    hPort : RTS_IEC_HANDLE;
    eRtsResult : RTS_IEC_RESULT;
    bReopenRequest : BOOL;
    GapTime : TIME := TIME#50ms;  (* Line quiet for this long ends a frame *)
    ReplyTimeout : TIME := TIME#1s0ms;  (* Nothing at all by now means no reply *)
    iState : INT;  (* 0 idle, 1 collecting, 2 judging *)
    eOutcome : E_RS485_STEP_STATE := E_RS485_STEP_STATE.IDLE;
    stStep : ST_RS485_STEP;  (* private copy: the caller's scratch is reused *)
    Data : A_RS485_READ_BUFFER;
    iRegCount : INT;
    abyTx : ARRAY[0..31] OF BYTE;  (* 9 + 2*8 for the largest FC16 *)
    iTxLen : INT;  (* payload before the wCrc *)
    abyRx : ARRAY[0..287] OF BYTE;
    udiRxCount : UDINT;
    abyFlush : ARRAY[0..287] OF BYTE;
    fbGap : TON;
    fbReplyTimer : TON;
    bRestartGap : BOOL;
    bRestartReply : BOOL;
    udiN : UDINT;  (* --- scratch ---------------------------------------------------------- *)
    pbyRx : POINTER TO BYTE;
    count : INT;
    iFirst : INT;
    iLast : INT;
    iFrameLen : INT;
    iK : INT;
    wCrc : WORD;
    uiEchoAddr : UINT;
    uiEchoValue : UINT;
    bDataValid : BOOL;
    stConfiguredSettings : SysCom.SysComSettings;  (* What Init bConfigured, saved so RestoreTuning can undo a commissioning sweep without the caller having to remember what it passed in. A sweep changes stSettings in place - that is the only way to reach the port - so the original has to live somewhere or it is gone. *)
    tConfiguredReplyTimeout : TIME;
    tConfiguredGapTime : TIME;
  END_VAR

            
          

METHOD ReadBuffer : POINTER TO A_RS485_READ_BUFFER
                  ReadBuffer := ADR(Data);

                
END_METHOD

METHOD Service : E_RS485_STEP_STATE
                  (* ---------------------------------------------------------------- the port *)
IF bReopenRequest THEN
	bReopenRequest := FALSE;
	IF PortOpen THEN
		SysCom.SysComClose(hPort);
	END_IF
	PortOpen	:= FALSE;
	PortError	:= FALSE;
	iState		:= 0;
	eOutcome		:= E_RS485_STEP_STATE.IDLE;
END_IF

IF bConfigured AND NOT PortOpen AND NOT PortError THEN
	hPort		:= SysCom.SysComOpen2(pSettings := ADR(stSettings), pSettingsEx := 0, pResult := ADR(eRtsResult));
	PortError	:= (hPort = RTS_INVALID_HANDLE OR eRtsResult <> 0);
	PortOpen	:= NOT PortError;
END_IF

(* Both timers are called unconditionally. A TON left with IN true while the
   iState machine is elsewhere goes on counting, and would then fire instantly
   on the next stStep. *)
fbGap(IN := (iState = 1) AND NOT bRestartGap, PT := GapTime);
fbReplyTimer(IN := (iState = 1) AND NOT bRestartReply, PT := ReplyTimeout);
bRestartGap		:= FALSE;
bRestartReply	:= FALSE;

(* ------------------------------------------------------- the stStep in flight *)
CASE iState OF

0:	(* Idle. OK and FAILED were each returned for exactly one cycle, by the
	   return at the bottom of the cycle that reached iState 2. *)
	eOutcome := E_RS485_STEP_STATE.IDLE;

1:	(* Collect until the line has been quiet for GapTime, which is how RTU
	   delimits a frame, or until the slave has clearly not answered at all. *)
	IF udiRxCount < SIZEOF(abyRx) THEN
		pbyRx := ADR(abyRx);
		pbyRx := pbyRx + udiRxCount;
		udiN := SysCom.SysComRead(hPort, pbyRx, SIZEOF(abyRx) - udiRxCount, 0, ADR(eRtsResult));
		IF udiN > 0 THEN
			udiRxCount		:= udiRxCount + udiN;
			bRestartGap	:= TRUE;
		END_IF
	END_IF

	(* A frame whose wCrc already checks out is complete by definition, so there
	   is nothing left to wait for. Waiting anyway costs about three task cycles
	   per stStep, and on a 200 ms task that is most of what a Modbus exchange
	   takes: measured at 1.87 s per stStep before this check, against roughly
	   100 ms of actual wire time at 9600 baud.

	   The silence timer stays as the fallback for everything that does not
	   frame cleanly - a partial reply, a burst of noise, a slave that answers
	   with something we cannot parse. *)
	count := UDINT_TO_INT(udiRxCount);
	IF count >= 5 AND THIS^.Frame() THEN
		iState := 2;
	ELSIF (udiRxCount > 0 AND fbGap.Q) OR fbReplyTimer.Q OR udiRxCount >= SIZEOF(abyRx) THEN
		iState := 2;
	END_IF

2:	THIS^.Judge();
	iState := 0;

END_CASE

Service := eOutcome;

                
END_METHOD

METHOD Start : BOOL
  VAR_INPUT
    pStep : POINTER TO ST_RS485_STEP;
  END_VAR
  VAR
    iI : INT;
    iQty : INT;
  END_VAR
                  Start := FALSE;

IF pStep = 0 OR NOT PortOpen OR iState <> 0 THEN
	RETURN;
END_IF

(* Private copy. The scheduler's stStep list is scratch that it reuses for the
   next device, so nothing may be read back out of it later - the echo checks
   below run against this copy. *)
stStep := pStep^;
iQty := UINT_TO_INT(stStep.Quantity);

CASE stStep.FunctionCode OF

3, 4:	(* read holding / read input registers *)
	IF iQty < 1 OR iQty > (DINT_TO_INT(UPPER_BOUND(Data, 1)) + 1) THEN
		RETURN;
	END_IF
	abyTx[0] := stStep.DeviceId;
	abyTx[1] := stStep.FunctionCode;
	abyTx[2] := UINT_TO_BYTE(SHR(stStep.Address, 8));
	abyTx[3] := UINT_TO_BYTE(stStep.Address AND 16#00FF);
	abyTx[4] := UINT_TO_BYTE(SHR(stStep.Quantity, 8));
	abyTx[5] := UINT_TO_BYTE(stStep.Quantity AND 16#00FF);
	iTxLen := 6;

6:	(* write single register: the value goes where the quantity would *)
	abyTx[0] := stStep.DeviceId;
	abyTx[1] := 16#06;
	abyTx[2] := UINT_TO_BYTE(SHR(stStep.Address, 8));
	abyTx[3] := UINT_TO_BYTE(stStep.Address AND 16#00FF);
	abyTx[4] := WORD_TO_BYTE(SHR(stStep.Data[0], 8));
	abyTx[5] := WORD_TO_BYTE(stStep.Data[0] AND 16#00FF);
	iTxLen := 6;

16:	(* write multiple registers: header, byte count, then the payload *)
	IF iQty < 1 OR iQty > (DINT_TO_INT(UPPER_BOUND(stStep.Data, 1)) + 1) THEN
		RETURN;
	END_IF
	abyTx[0] := stStep.DeviceId;
	abyTx[1] := 16#10;
	abyTx[2] := UINT_TO_BYTE(SHR(stStep.Address, 8));
	abyTx[3] := UINT_TO_BYTE(stStep.Address AND 16#00FF);
	abyTx[4] := UINT_TO_BYTE(SHR(stStep.Quantity, 8));
	abyTx[5] := UINT_TO_BYTE(stStep.Quantity AND 16#00FF);
	abyTx[6] := INT_TO_BYTE(iQty * 2);
	FOR iI := 0 TO iQty - 1 DO
		abyTx[7 + 2 * iI] := WORD_TO_BYTE(SHR(stStep.Data[iI], 8));
		abyTx[8 + 2 * iI] := WORD_TO_BYTE(stStep.Data[iI] AND 16#00FF);
	END_FOR
	iTxLen := 7 + 2 * iQty;

ELSE
	(* Refused, not guessed at. Guessing is precisely the bug this replaces:
	   every function code used to be framed from the read fields, so an FC6
	   write went out as "write register 0 := 0" and its echoed reply was then
	   parsed as though byte 2 were a length. *)
	RETURN;

END_CASE

(* Anything still in the receive buffer belongs to the previous exchange and
   would otherwise be collected as this one's reply. *)
udiN := SysCom.SysComRead(hPort, ADR(abyFlush), SIZEOF(abyFlush), 0, ADR(eRtsResult));

wCrc := THIS^.Crc16(pBuf := ADR(abyTx), Len := iTxLen);
abyTx[iTxLen]		:= WORD_TO_BYTE(wCrc AND 16#00FF);
abyTx[iTxLen + 1]	:= WORD_TO_BYTE(SHR(wCrc, 8));

SysCom.SysComWrite(hPort, ADR(abyTx), INT_TO_UDINT(iTxLen + 2), 100, ADR(eRtsResult));

udiRxCount			:= 0;
iRegCount		:= 0;
bRestartGap		:= TRUE;
bRestartReply	:= TRUE;
eOutcome			:= E_RS485_STEP_STATE.BUSY;
iState			:= 1;
Start			:= TRUE;

                
END_METHOD

METHOD Judge
  VAR
    iBytecount : INT;
    iI : INT;
    bGotFrame : BOOL;
  END_VAR
                  count		:= UDINT_TO_INT(udiRxCount);
bGotFrame	:= THIS^.Frame();

(* Leading glitch bytes are the slave's driver enabling onto an undriven pair,
   trailing ones its releasing. Both are normal on this hardware. *)
IF iFirst > 0 THEN
	LeadNulls := LeadNulls + 1;
END_IF
IF bGotFrame AND iLast < count THEN
	TrailNulls := TrailNulls + 1;
END_IF

iFrameLen	:= iLast - iFirst;
iRegCount	:= 0;
bDataValid		:= FALSE;

IF count = 0 OR (count - iFirst) = 0 THEN
	NoReply := NoReply + 1;

ELSIF (count - iFirst) < 5 THEN
	ShortFrame := ShortFrame + 1;

ELSIF NOT bGotFrame THEN
	CrcFail := CrcFail + 1;

	(* Capture what actually arrived. Two theories about these failures have now
	   been wrong - leading glitch bytes, then a framer that could not
	   resynchronise - and both were argued from counters rather than from
	   bytes. A counter says a frame did not check out; it cannot say whether
	   what arrived was half a reply, two replies, an echo, or noise. Decimal
	   rather than hex because there is no hex helper in scope and the point is
	   to read it off an MQTT topic, not to look pretty. *)
	LastFailLen := udiRxCount;

	(* Whose window this landed in. Without it the bytes are unattributable, and
	   a frame that looks like somebody else's request is exactly the case that
	   needs telling apart from a mangled reply. *)
	LastFailAddr := stStep.DeviceId;
	LastFailFunc := stStep.FunctionCode;

	LastFailBytes := '';
	FOR iI := 0 TO count - 1 DO
		IF iI >= 24 THEN
			EXIT;
		END_IF
		LastFailBytes := CONCAT(LastFailBytes, BYTE_TO_STRING(abyRx[iI]));
		LastFailBytes := CONCAT(LastFailBytes, ' ');
	END_FOR

ELSIF abyRx[iFirst] <> stStep.DeviceId THEN
	(* Well formed, intact, and not ours. On a shared bus that is somebody
	   else's traffic; on this one it means the reply was mis-framed. *)
	BadAddress := BadAddress + 1;

ELSIF abyRx[iFirst + 1] = (stStep.FunctionCode OR 16#80) THEN
	Exceptions		:= Exceptions + 1;
	LastException	:= abyRx[iFirst + 2];

ELSIF abyRx[iFirst + 1] <> stStep.FunctionCode THEN
	BadFunction := BadFunction + 1;

ELSE
	CASE stStep.FunctionCode OF

	3, 4:	(* addr, fc, byte count, data, crc16 *)
		iBytecount := BYTE_TO_INT(abyRx[iFirst + 2]);
		IF iBytecount < 2 OR iBytecount > (iFrameLen - 5) THEN
			ShortFrame := ShortFrame + 1;
		ELSE
			iRegCount := iBytecount / 2;
			IF iRegCount > (DINT_TO_INT(UPPER_BOUND(Data, 1)) + 1) THEN
				iRegCount := DINT_TO_INT(UPPER_BOUND(Data, 1)) + 1;
			END_IF
			(* Registers are big-endian on the wire, which is the order
			   F_SWAP_WORDS_TO_REAL expects at the far end. *)
			FOR iI := 0 TO iRegCount - 1 DO
				Data[iI] := SHL(BYTE_TO_WORD(abyRx[iFirst + 3 + 2 * iI]), 8)
				           OR BYTE_TO_WORD(abyRx[iFirst + 4 + 2 * iI]);
			END_FOR
			Ok		:= Ok + 1;
			bDataValid	:= TRUE;
		END_IF

	6:	(* The reply is the request echoed back. There is no byte count in it,
		   and reading byte 2 as one - which is what this code did for every
		   function code before - reads an address high byte as a length. *)
		IF iFrameLen < 8 THEN
			ShortFrame := ShortFrame + 1;
		ELSE
			uiEchoAddr	:= SHL(BYTE_TO_UINT(abyRx[iFirst + 2]), 8) OR BYTE_TO_UINT(abyRx[iFirst + 3]);
			uiEchoValue	:= SHL(BYTE_TO_UINT(abyRx[iFirst + 4]), 8) OR BYTE_TO_UINT(abyRx[iFirst + 5]);
			IF uiEchoAddr <> stStep.Address OR uiEchoValue <> WORD_TO_UINT(stStep.Data[0]) THEN
				(* The slave acknowledged something other than what was asked.
				   Never report this as success: a read-after-write would then
				   publish a confirmation for a write that did not happen. *)
				BadEcho := BadEcho + 1;
			ELSE
				Ok		:= Ok + 1;
				bDataValid	:= TRUE;
			END_IF
		END_IF

	16:	(* addr, 16, start address, quantity written, crc16 *)
		IF iFrameLen < 8 THEN
			ShortFrame := ShortFrame + 1;
		ELSE
			uiEchoAddr	:= SHL(BYTE_TO_UINT(abyRx[iFirst + 2]), 8) OR BYTE_TO_UINT(abyRx[iFirst + 3]);
			uiEchoValue	:= SHL(BYTE_TO_UINT(abyRx[iFirst + 4]), 8) OR BYTE_TO_UINT(abyRx[iFirst + 5]);
			IF uiEchoAddr <> stStep.Address OR uiEchoValue <> stStep.Quantity THEN
				BadEcho := BadEcho + 1;
			ELSE
				Ok		:= Ok + 1;
				bDataValid	:= TRUE;
			END_IF
		END_IF

	END_CASE
END_IF

IF bDataValid THEN
	eOutcome := E_RS485_STEP_STATE.OK;
ELSE
	eOutcome := E_RS485_STEP_STATE.FAILED;
END_IF

                
END_METHOD

METHOD Frame : BOOL
  VAR
    iTries : INT;
  END_VAR
                  (* Find the frame inside what has been collected. Sets `iFirst` and `iLast`, and
   returns whether the bytes between them check out.

   Counts nothing, changes no iState beyond those two indices, and is safe to
   call every cycle - which is the point. Service uses it to notice that a frame
   is already complete instead of waiting out the silence, and Judge uses it to
   decide what it is looking at.

   This RESYNCHRONISES rather than merely trimming a leading run of nulls, and
   that distinction is the whole reason it was rewritten. Trimming nulls handles
   the driver-enable glitch this hardware produces, and nothing else: put any
   non-zero byte in front of the reply and every wCrc trial fails, because the
   window always started at that byte. Measured on a DFRobot SEN0492, one reply
   in three was being thrown away that way - bytes present, LeadNulls climbing,
   CrcFail climbing, and the sensor answering perfectly well the whole time.

   Three things put a non-zero byte in front of a reply, and all of them are
   ordinary rather than exotic:
     - a slave that echoes the request before answering, which is documented
       behaviour for the SEN0492 and reported for others;
     - a byte left over from the previous exchange that arrived after Start
       flushed the port;
     - two replies collected into one window, when a slave answers late enough
       to land inside the next poll.
   All three are cured by asking "does a valid frame start HERE?" at every
   plausible offset instead of assuming the answer is offset zero.

   The search is anchored on the slave address rather than sweeping blindly,
   which keeps the number of wCrc trials small and, more importantly, keeps the
   chance of a coincidental wCrc match negligible. *)
Frame	:= FALSE;
iFirst	:= 0;

WHILE NOT Frame AND iFirst <= (count - 5) DO

	(* Only a byte that could be this slave's reply is worth testing. *)
	IF abyRx[iFirst] = stStep.DeviceId THEN

		(* Trailing bytes are removed by asking the wCrc rather than by assuming
		   a trailing 00 is noise. It usually is - but a frame whose wCrc high
		   byte is genuinely 00 turns up about once in 256, and blindly trimming
		   it turned a perfectly good reply into a wCrc failure. *)
		iLast	:= count;
		iTries	:= 0;

		WHILE NOT Frame AND iTries < 4 AND (iLast - iFirst) >= 5 DO
			IF THIS^.Crc16(pBuf := ADR(abyRx[iFirst]), Len := iLast - iFirst) = 0 THEN
				Frame := TRUE;
			ELSE
				iLast	:= iLast - 1;
				iTries	:= iTries + 1;
			END_IF
		END_WHILE

	END_IF

	IF NOT Frame THEN
		iFirst := iFirst + 1;
	END_IF

END_WHILE

(* Nothing framed. Leave `iFirst` and `iLast` describing the buffer the way the
   old null-trimming did, because Judge classifies the failure from them: a
   `iFirst` left pointing near the end would turn a wCrc failure into a reported
   short frame, which is a worse diagnosis than the one it replaces. *)
IF NOT Frame THEN
	iFirst := 0;
	WHILE iFirst < count AND abyRx[iFirst] = 0 DO
		iFirst := iFirst + 1;
	END_WHILE
	iLast := count;
END_IF

                
END_METHOD

METHOD Crc16 : WORD
  VAR_INPUT
    pBuf : POINTER TO BYTE;
    Len : INT;
  END_VAR
  VAR
    iI : INT;
    iB : INT;
    wAcc : WORD;
    pbyP : POINTER TO BYTE;
  END_VAR
                  (* Modbus RTU CRC16: polynomial 16#A001, seed 16#FFFF, transmitted low byte
   iFirst. A whole bDataValid frame including its own wCrc therefore checksums to zero,
   which is how a received frame is judged - no need to know where the data
   ends before deciding whether it is intact. *)
wAcc := 16#FFFF;
pbyP := pBuf;

FOR iI := 0 TO Len - 1 DO
	wAcc := wAcc XOR BYTE_TO_WORD(pbyP[iI]);
	FOR iB := 0 TO 7 DO
		IF (wAcc AND 16#0001) <> 0 THEN
			wAcc := SHR(wAcc, 1) XOR 16#A001;
		ELSE
			wAcc := SHR(wAcc, 1);
		END_IF
	END_FOR
END_FOR

Crc16 := wAcc;

                
END_METHOD

METHOD Reopen
                  (* Close and re-open on the next Service. Clears PortError too, so a port that
   failed to open at boot - a controller still coming up, say - can be retried
   without a download. *)
bReopenRequest := TRUE;

                
END_METHOD

METHOD Init
  VAR_INPUT
    Port : SysCom.SYS_COM_PORTS;  (* Which serial port. Only SYS_COMPORT1 is exposed by the PFC200 runtime - COM2, COM3 and COM4 were all tried in #182 and every one of them failed to open. *)
    Baudrate : UDINT;  (* Bits per second. 9600 for every device this project has met. *)
    Parity : SysCom.SYS_COM_PARITY;
    StopBits : SysCom.SYS_COM_STOPBITS;  (* Modbus specifies two stop bits with no parity, but every device tested here answers on one. Ask the device, not the standard. *)
    ReplyTimeout : TIME;  (* Nothing at all by now means no reply. Zero keeps the default of one second. *)
    GapTime : TIME;  (* Line quiet for this long ends a frame - the 3.5-character silence RTU actually specifies, rounded up to something a 200 ms task can see. Zero keeps the default of 50 ms. *)
  END_VAR
                  (* stSettings are assigned here rather than in a declaration initialiser. A value
   inside an existing structured initialiser cannot be changed from a script -
   the compiler goes on reading the stored structValue - and having them in code
   means Reopen can bring the port back up with different stSettings from an
   online session. *)
stSettings.sPort			:= Port;
stSettings.ulBaudrate		:= Baudrate;
stSettings.byParity		:= Parity;
stSettings.byStopBits		:= StopBits;
stSettings.ulTimeout		:= 0;
stSettings.ulBufferSize	:= 256;

IF ReplyTimeout > T#0S THEN
	THIS^.ReplyTimeout := ReplyTimeout;
END_IF
IF GapTime > T#0S THEN
	THIS^.GapTime := GapTime;
END_IF

(* Remember all of it, so Retune can wander off and RestoreTuning can come back
   without the caller repeating itself. Taken after the defaults above have been
   applied, so what is saved is what the port is actually running. *)
stConfiguredSettings		:= stSettings;
tConfiguredReplyTimeout	:= THIS^.ReplyTimeout;
tConfiguredGapTime		:= THIS^.GapTime;

bConfigured := TRUE;

(* Re-open if the port was already up, so calling Init twice is not a silent
   no-op with the old stSettings still in force. *)
bReopenRequest := PortOpen;

                
END_METHOD

METHOD Registers : INT
                  Registers := iRegCount;

                
END_METHOD

(* Re-open the bus at a different setting, keeping everything Init bConfigured that is not named here. Sentinels rather than optional parameters, because a caller sweeping a bus needs to vary one field at a time: 0 for a rate or a time and 255 for framing all mean "leave it alone". This is what makes commissioning possible at all - a device that ships on the wrong baud rate has to be hunted for at rates the bus does not use - and it belongs here rather than at the caller: nothing outside can see the port stSettings, and nothing outside should have to know the port, parity or buffer size in order to change one field. Returns FALSE from a transport that cannot be re-tuned. A sweep must then give up rather than probe at a setting it only thinks it applied. *)
METHOD Retune : BOOL
  VAR_INPUT
    Baudrate : UDINT;  (* 0 keeps the bConfigured rate *)
    StopBitsRaw : BYTE;  (* 255 keeps the bConfigured framing *)
    ReplyTimeout : TIME;  (* T#0S keeps the bConfigured timeout *)
    GapTime : TIME;  (* T#0S keeps the bConfigured fbGap *)
  END_VAR
                  (* One field at a time, which is what a sweep needs: everything not named here
   stays as Init bConfigured it. Takes effect on the next Service, like Reopen. *)
IF NOT bConfigured THEN
	Retune := FALSE;
	RETURN;
END_IF

IF Baudrate > 0 THEN
	stSettings.ulBaudrate := Baudrate;
END_IF
IF StopBitsRaw <> 255 THEN
	stSettings.byStopBits := StopBitsRaw;
END_IF
IF ReplyTimeout > T#0S THEN
	THIS^.ReplyTimeout := ReplyTimeout;
END_IF
IF GapTime > T#0S THEN
	THIS^.GapTime := GapTime;
END_IF

Reopen();
Retune := TRUE;

                
END_METHOD

(* Put the bus back to exactly what Init bConfigured, however far a sweep wandered. Kept as the transport's own saved copy rather than re-derived, so a caller does not have to remember what it passed to Init in order to hand it back - and so a sweep that ends early, or fails, still leaves a bus the rest of the devices can use. *)
METHOD RestoreTuning
                  (* Whatever a sweep did to stSettings, this is the way back. Reopen rather than an
   immediate close: the port is only ever touched from Service, so that a caller
   cannot pull the bus out from under a frame in flight. *)
IF NOT bConfigured THEN
	RETURN;
END_IF

stSettings		:= stConfiguredSettings;
ReplyTimeout	:= tConfiguredReplyTimeout;
GapTime			:= tConfiguredGapTime;

Reopen();

                
END_METHOD

(* Bytes in the iLast receive window, framed or not. The counter that matters when a device answers nothing at all. Zero bytes at every setting is a bus with nothing on it; bytes that arrive and never frame are a device that is present and being read wrongly - or a pair that is the wrong way round. That distinction is invisible from anywhere else, and it is the one that says whether to keep sweeping stSettings or go and look at the wiring. *)
METHOD LastRxCount : UDINT
                  LastRxCount := udiRxCount;

                
END_METHOD
END_FUNCTION_BLOCK

{attribute 'do_checks_for_implicit_code'}
PROGRAM PRG_MAIN
  VAR
    fbDiPb001 : FB_INPUT_PUSHBUTTON_MQTT := (FriendlyName := 'Button number 001');  (* Every MQTT block below now wires itself from GVL_MQTT on its first cyclic call. Setting FriendlyName is what enables that, and it is the only thing a normal instance has to say. The InitMqtt / InitMqttDiscovery* calls that used to live in MAIN_INIT are gone. EntityType is only needed where a block can announce as more than one Home Assistant platform and you do not want its default. Both switched outputs below are announced as lights, which is what they announced before this refactor - leaving that out would silently orphan their retained light/.../config topics and create switch entities instead. INPUT FUNCTION BLOCKS *)
    fbDiPb002 : FB_INPUT_PUSHBUTTON_DIMMER_MQTT := (FriendlyName := 'Button number 002');
    fbAiRtdUnwired : FB_INPUT_TEMPERATURE_RTD_MQTT;  (* ANALOG INPUT FUNCTION BLOCKS No RTD module on this bench, so no channel to read. This instance is declared and called anyway, unwired, because a function block that nothing instantiates is never compiled - it would go on exporting and reading as supported while a change to FB_MQTT_BASE or the discovery device quietly broke it. FriendlyName is empty, so it wires nothing and announces nothing. Put a module back and this is where the real instances go: one per channel, Raw wired to the channel word, FriendlyName set, and ProcessImageValid := Pfc200Bus.xConfigFinished. See docs/AnalogInputs/UsingRTDSensors.md. *)
    fbDoBin001 : FB_OUTPUT_BINARY_MQTT := (FriendlyName := 'light number 2', EntityType := E_MQTT_ENTITY.Light);  (* OUTPUT FUNCTION BLOCKS *)
    fbDoBistable001 : FB_OUTPUT_BISTABLE_MQTT := (FriendlyName := 'light number 1', EntityType := E_MQTT_ENTITY.Light);
    fbDoCover001 : FB_OUTPUT_COVER_MQTT := (FriendlyName := 'cover number 001');  (* COVER FUNCTION BLOCKS FB_init args are (T_LOCKOUT, T_UD): 1s between direction changes, 20s to travel fully up or down. *)
    fbDoCover002 : FB_OUTPUT_COVER_POSITION_MQTT := (FriendlyName := 'cover number 002');  (* The same shutter hardware, but with a position slider in Home Assistant. Travel times are inputs rather than FB_init arguments here - they are the one number on a cover somebody always ends up tuning, and an FB_init argument cannot be revised by tooling. *)
    fbAoDimmer001 : FB_OUTPUT_DIMMER_MQTT := (FriendlyName := '001. Office strip cold');  (* E_DIMMER FUNCTION BLOCKS NOTE: this instance never had InitMqtt called before this refactor - only ConfigureFunctionBlock and InitMqttDiscovery, and the latter short-circuited because InitMqttDone stayed FALSE. It therefore had no MQTT topic, no Home Assistant entity and no control at all. Naming it here fixes that, which means this instance starts publishing for the first time. *)
    wTestOUT : WORD;
    bKbusEnableIoCheck : BOOL := FALSE;  (* K-BUS CONTROL Pfc200Bus is the K-bus driver instance the device tree declares - an IoDrvPfc200, which offers exactly one input and one property worth reaching from IEC code. Both are wired in READ_PUSHBUTTONS. Neither is written by anything in this project. They are here to be set by hand from an online view, which is the only way they are ever meant to be used. Hands the K-bus transmission cycle to the PFC firmware instead of CODESYS, which is what lets WAGO-I/O-CHECK reach the modules over the service cable while the runtime keeps running. Set it TRUE, pulse bKbusRestart to make it take effect, configure the modules, then put it back to FALSE and pulse bKbusRestart again - otherwise CODESYS never gets its bus cycle back. *)
    bKbusRestart : BOOL;  (* A rising edge restarts the K-bus. On its own - with bKbusEnableIoCheck left FALSE - that is the recovery for a bus that has stopped exchanging process data; the I/O LED should come back to steady green. *)
  END_VAR

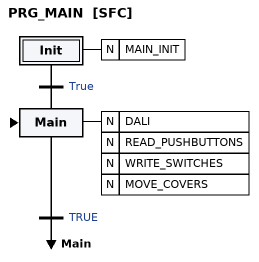
INITIAL_STEP Init:
  MAIN_INIT(N);
END_STEP
TRANSITION FROM Init TO Main
  := True;
END_TRANSITION
STEP Main:
  DALI(N);
  READ_PUSHBUTTONS(N);
  WRITE_SWITCHES(N);
  MOVE_COVERS(N);
END_STEP
TRANSITION FROM Main TO Main
  := TRUE;
END_TRANSITION

ACTION MOVE_COVERS:
                        (* fbDoCover001 keeps the relays it always had. The position-capable block gets
   DO_005 and DO_006, freed in HVAC_RUN for exactly this - two LEDs on the second
   output module that can be watched while the cover is commanded from Home
   Assistant, which is what makes the position logic verifiable at a glance.

   One writer per coil, in one task. DO_005..DO_008 used to be written from
   HvacTask, and a second writer here would have made both meaningless without the
   compiler saying a word. *)
fbDoCover001(
	TOGGLE:=fbDiPb001.P_LONG,
	MU=>DO_003,
	MD=>DO_004
);

fbDoCover002(
	T_TravelUp := T#20S,
	T_TravelDown := T#20S,
	MU => DO_005,
	MD => DO_006
);

                      
END_ACTION

ACTION READ_PUSHBUTTONS:
                        fbDiPb001(PB:= DI_001); (* Provide the input FB the correct phyical input to validate each cyclus *)
fbDiPb002(PB:= DI_002);
(* Called so the block is compiled, not to read anything: see its declaration.
   Raw is a literal because there is no channel word on this bench, and with
   ProcessImageValid left FALSE the block reports the reading as invalid, which
   is exactly what an unwired input is. *)
fbAiRtdUnwired(Raw := 0);


(* K-BUS CONTROL. Written every cycle so that setting either flag in an online
   view is enough; see their declarations for what they do and in which order.
   Pfc200Bus() is called explicitly because that is what reads xRestart - the
   implicit bus cycle call does not. *)
Pfc200Bus.EnableIoCheck := bKbusEnableIoCheck;
Pfc200Bus.xRestart := bKbusRestart;
Pfc200Bus();

                      
END_ACTION

ACTION MAIN_INIT:
                        (* MQTT wiring no longer lives here.

   Every block that extends FB_MQTT_BASE now wires itself from GVL_MQTT on
   its first cyclic call and announces itself to Home Assistant, driven by the
   FriendlyName set on its declaration above. What remains in this action is the
   behavioural configuration that genuinely is per-instance and is not MQTT, which
   is now only the E_DIMMER's timings. *)

(* ALTER THE E_DIMMER OUTPUT DEFAULT BEHAVIOR *)
fbAoDimmer001.ConfigureFunctionBlock(
	T_Debounce:=T#10MS,
	T_Reconfig:=T#10S,
	T_On_Max:=T#0S,
	T_Dimm_Start:=T#400MS,
	T_Dimm:=T#3S,
	Min_On:=50,
	Max_On:=255,
	Soft_Dimm:=TRUE,
	Rst_Out:=FALSE,
	OUT_LinearScaleMin:=11000,
	OUT_LinearScaleMax:=32767
);


(* Cover timings now travel through FB_init at the instance declaration. *)


(* DALI *)
(*
FB_DALI_1_ADR0.InitMqtt(MQTTPublishPrefix:= ADR(GVL_MQTT.MqttPubDimmerPrefix),
	MQTTSubscribePrefix:= ADR(GVL_MQTT.MqttSubDimmerPrefix),
	pMqttPublishQueue := ADR(GVL_MQTT.fbMqttPublishQueue),
	pMqttCallbackCollector := ADR(GVL_MQTT.collector_FB_DIMMER_MQTT)
);

FB_DALI_1_ADR0.InitMqttDiscovery(ADR(GVL_MQTT.PLC_Device), 'Keuken');
*)

GVL_MQTT.PLC_Device.SendLogMessage('Init finished', 'MAIN_INIT');

                      
END_ACTION

ACTION WRITE_SWITCHES:
                        fbDoBin001(OUT	=>		DO_001,										(* couple the function block to the physical output *)
	PRIO_HIGH				:=FALSE,  									(* brings the output high regardless of other input values *)
	PRIO_LOW				:=FALSE, 									(* brings the output low regardless of other input values. NOTE: PRIO_HIGH overrules PRIO_LOW input *)
	TOGGLE					:=fbDiPb001.SINGLE 						(* for toggling the output *)	
);

fbAoDimmer001(
	SINGLE:=fbDiPb001.SINGLE,
	LONG:=fbDiPb001.LONG, 
	P_LONG:=fbDiPb001.P_LONG, 
	Q_OUT => wTestOUT,
	SET:=  fbDiPb001.DOUBLE,
	VAL:=125
);

fbDoBistable001();
                      
END_ACTION

ACTION DALI:
                        // Run the master before anything else
(*
M1_DALIMASTER(
	bPortDALI:=1,
	I_Port:=IoConfig_Globals.DALI_MULTI_MASTER_MODULE);
	
// Run individual DALI FB
FB_DALI_1_ADR0(
	BALLAST := GVL_DALI.M1_Light1,
	TOGGLE := fbDiPb002.SINGLE,
	P_LONG := fbDiPb002.P_LONG,
	STATUS_LED => DO_002);
	*)
                      
END_ACTION
END_PROGRAM

PROGRAM PRG_DMX_SEND
  VAR
    iUniverse : INT := 1;
    IP_CONTROL2 : oscat_network.IP_CONTROL2;
    IP_C : oscat_network.IP_C;
    stSBuf1 : oscat_network.NETWORK_BUFFER_SHORT;
    stRBuf1 : oscat_network.NETWORK_BUFFER_SHORT;
    bErrorSend : BOOL := FALSE;
    iI : INT;
    init : BOOL;
    start : INT;
    size : INT;
    iStep : INT := 0;
    fbErrorTrig : Standard.R_TRIG;  (* Rate-limits the connection-error log to one message per error, instead of one per scan of a freewheeling task. *)
  END_VAR

                    IF init = FALSE THEN
	init := TRUE;
	//https://art-net.org.uk/how-it-works/streaming-packets/artdmx-packet-definition/
	(* Write DMX header character in the buffer *) 
	stSBuf1.BUFFER [0]:= BYTE#16#41; // A
	stSBuf1.BUFFER [1]:= BYTE#16#72; // R	
	stSBuf1.BUFFER [2]:= BYTE#16#74; // T
	stSBuf1.BUFFER [3]:= BYTE#16#2D; // -
	stSBuf1.BUFFER [4]:= BYTE#16#4E; // N
	stSBuf1.BUFFER [5]:= BYTE#16#65; // E
	stSBuf1.BUFFER [6]:= BYTE#16#74; // T
	stSBuf1.BUFFER [7]:= BYTE#16#00; // 0 zero
	
	stSBuf1.BUFFER [8]:= BYTE#16#00;	// Opcode ArtDMX (0x5000) little endian
	stSBuf1.BUFFER [9]:= BYTE#16#50; // Opcode ArtDMX (0x5000) little endian
	
	stSBuf1.BUFFER [10]:= BYTE#16#00; // Protocol Version Hi (0)
	stSBuf1.BUFFER [11]:= BYTE#16#0E; // Protocol Version Lo (14)
	
	stSBuf1.BUFFER [12]:= BYTE#16#00; // Sequence
	stSBuf1.BUFFER [13]:= BYTE#16#00; // Physical
	
	stSBuf1.BUFFER [16]:= BYTE#16#02; // Length Hi
	stSBuf1.BUFFER [17]:= BYTE#16#00; // Length Lo (2 to 512, even)
	(* the DMX channels that are next have already been written to the buffer *) 
	
	IF iUniverse = 1 THEN
		stSBuf1.BUFFER [14]:= BYTE#16#01; // iUniverse little endian
		stSBuf1.BUFFER [15]:= BYTE#16#00; // iUniverse little endian
	END_IF
	IF iUniverse = 2 THEN
		stSBuf1.BUFFER [14]:= BYTE#16#02; // iUniverse little endian
		stSBuf1.BUFFER [15]:= BYTE#16#00; // iUniverse little endian
	END_IF
END_IF;


size := 512+18;
FOR iI:= 0 TO 511 DO (* check whether the DMX values ​​in the global variable have changed *)
	(* One convention, and it is asserted here: GVL_DMX.DMX.BUFFER[c - 1] holds
	   DMX channel c, which is what FB_OUTPUT_DIMMER_DMX_MQTT writes. An ArtDmx
	   packet carries its 18-byte header and then channel 1 at data offset 0, so
	   buffer index iI goes to BUFFER[iI + 18] and nothing shifts on the way.

	   This read used to be BUFFER[iI + 2] against a block writing BUFFER[c - 1]:
	   channel c lit slot c - 2, and channels 1 and 2 could not be reached at all
	   because no iteration ever read buffer index 0 or 1. *)
	IF stSBuf1.BUFFER[iI+18] <> GVL_DMX.DMX.BUFFER[iI] THEN
   		stSBuf1.BUFFER[iI+18]:= GVL_DMX.DMX.BUFFER[iI];
		iStep := 1;
	END_IF
END_FOR



fbErrorTrig(CLK := IP_C.ERROR <> 0);

CASE iStep OF
	0:
		//passive
	
	1:
		IP_C.C_MODE := 1; (* Mode: UDP+ACTIVE+Port+IP *)
		IP_C.C_ENABLE := TRUE; (* Release connection *)
		IP_C.TIME_RESET := TRUE; (*Reset TIME monitoring * *)
		IP_C.R_OBSERVE := TRUE; (* Monitor data receive *)
		stRBuf1.SIZE:= 0; (* Reset Home length *)
		IP_C.C_IP:= oscat_network.IP4_DECODE (GVL_DMX.IP);
		IP_C.C_PORT:= WORD#6454;
		
		stSBuf1.SIZE := size;
		iStep:=2;
		
	2:
		IP_CONTROL2 (TIME_OUT:= T#1S, IP_C:= IP_C, S_BUF:= stSBuf1, R_BUF:= stRBuf1);
		
		IF IP_C.ERROR <> 0  THEN
			iStep:=666;
		END_IF
	666:		
     	PFC.SetLed(which:=PFC.LED.U3, how:=PFC.LedState.BLINK_RED);
		IF fbErrorTrig.Q AND IP_C.ERROR = 33554432 THEN
		GVL_MQTT.PLC_Device.SendLogMessage(CONCAT('ERROR|DMX has a connection error ', DWORD_TO_STRING(IP_C.ERROR)));
		
		END_IF;
		
		bErrorSend := TRUE;
		stRBuf1.SIZE := 0;
		IP_C.C_ENABLE:= FALSE; (* Enable connection establishment *) 
		IP_C.TIME_RESET:= FALSE;
		init:=FALSE;
		(* Leave the error state. Without this the branch re-ran every scan; init is
		   FALSE so the header is rebuilt, and the change-detect loop re-arms iStep. *)
		iStep := 0;
	ELSE
	  iStep := 0;
END_CASE



// Check IP_C1.error
// 33554432 = 0x02000000
// Initialization of the socket interface failed (only WinNT).
// code = 0x 02 00 00 00 (hexadecimal)
//           !   !    ! 
//           !   !    Receive error 
//           !   Send error
//           Connect error

                  
END_PROGRAM

{attribute 'do_checks_for_implicit_code'}
PROGRAM PRG_MQTT
  VAR
    MQTT_IN_OUT : MQTT.MQTT_IN_OUT;
    stMQTTInfo : MQTT.MQTT_INFO;
    stMQTTBirthMessage : ST_MQTT_MESSAGE;
    fbMQTTBirthHartbeat : OSCAT_BASIC.GEN_PULSE;
    fbMQTTConnectTrigger : Standard.R_TRIG;
    bBrokerHealthy : BOOL;  (* Broker health as U1 reports it: an MQTT session AND the broker reachable. *)
    bLedShowsHealthy : BOOL;  (* What U1 is currently showing, so SetLed is called only when it changes. FALSE after a cold reset, which is the state MQTT_INIT puts the LED in. *)
    bMQTTPublishBirth : BOOL := TRUE;
    fbMQTTBirthPublisher : FB_MQTT_PUBLISH_WORKER;
    initMqtt : BOOL;  (* variables for MQTT setup *)
    udiIcounter : UDINT;
    afbPublishers : ARRAY[0..(cudiPublishers - 1)] OF FB_MQTT_PUBLISH_WORKER;  (* variables for MQTT publishing. The pool size is a constant and the array is sized from it: they used to be two literals that had to agree by hand, and the count was a plain VAR - writable from an online view, where setting it to 0 made FOR udiI := 0 TO (count - 1) underflow UDINT to 4294967295 and walk off the end of the array. *)
    udiI : UDINT;  (* variables to work with Mqttbuffer *)
    fbSubscriberFbOutputSwitchMqtt : MQTT.MQTTSubscribe;  (* variables for MQTT subscribing *)
    fbSubscriberFbOutputCoverMqtt : MQTT.MQTTSubscribe;
    fbSubscriberFbDimmerMqtt : MQTT.MQTTSubscribe;
    fbSubscriberFbRs485Mqtt : MQTT.MQTTSubscribe;
    fbSubscriberFbHvacMqtt : MQTT.MQTTSubscribe;
  END_VAR
  VAR CONSTANT
    cudiPublishers : UDINT := 40;
  END_VAR
  VAR
    fbSessionDrop : F_TRIG;  (* a session ended: one will at the broker *)
    fbSessionStable : TON;  (* connected long enough to count as working *)
    fbMqttStalled : TON;  (* nothing has worked for a long time *)
    fbMqttCoolDown : TON;  (* how long ENABLE stays off after a stall *)
    bMqttEnable : BOOL := TRUE;  (* drives the client's ENABLE pin *)
    bSessionWasStable : BOOL;  (* so the log fires once per recovery *)
    tMqttRest : TIME := GVL_MQTT.tMqttReconnectRestMin;
    udiSessionDrops : UDINT;  (* drops since the last stable session *)
    udiSessionDropsTotal : UDINT;  (* drops since the application started *)
    udiMqttCoolDowns : UDINT;  (* stalls that needed ENABLE cycling *)
  END_VAR

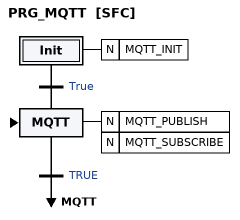
INITIAL_STEP Init:
  MQTT_INIT(N);
END_STEP
TRANSITION FROM Init TO MQTT
  := True;
END_TRANSITION
STEP MQTT:
  MQTT_PUBLISH(N);
  MQTT_SUBSCRIBE(N);
END_STEP
TRANSITION FROM MQTT TO MQTT
  := TRUE;
END_TRANSITION

ACTION MQTT_PUBLISH:
                        (* allow the device to do its work *)
GVL_MQTT.PLC_Device();

(* The MQTT client reports its own state on an output, so copy it in before anything
   looks at it. Nothing populated stMQTTInfo before this line existed, which is why
   MQTT_CONNECTED was permanently FALSE: no edge could ever fire, so the U1 LED never
   went green and the birth message was left to the heartbeat alone. *)
stMQTTInfo := MQTT_IN_OUT.clientFB.MQTT_INFO;

(* Healthy means the client has a session AND the broker is really reachable, and the
   second half is not redundant: MQTT_CONNECTED does not notice a pulled network
   cable. TCP has nothing to report until a retransmit finally gives up, so the client
   holds a dead socket open for minutes and goes on claiming a session. Verified on
   the bench: LAN cable out, MQTT_CONNECTED still TRUE, U1 still green.
   GVL_MQTT.bBrokerReachable is an ICMP check owned by the Ping task. *)
bBrokerHealthy := stMQTTInfo.MQTT_CONNECTED AND GVL_MQTT.bBrokerReachable;

(* U1 makes broker health readable from the cabinet without a laptop: steady green
   while it is healthy, blinking red while it is not.

   Written only when it changes, because SetLed is a runtime call - but from a
   remembered state rather than from a pair of edge detectors, so there is one code
   path instead of two. Two is how this was broken before: the falling-edge detector
   was called once, from MQTT_INIT, so its Q could never become TRUE and the LED
   could never go red, while the rising-edge half looked perfectly fine.
   bLedShowsHealthy also reports what the LED is showing, which a one-cycle Q cannot,
   so a test can read the colour back. *)
IF bBrokerHealthy <> bLedShowsHealthy THEN
	IF bBrokerHealthy THEN
		PFC.SetLed(which := PFC.LED.U1, how := PFC.LedState.STATIC_GRN);
	ELSE
		PFC.SetLed(which := PFC.LED.U1, how := PFC.LedState.BLINK_RED);
	END_IF
	bLedShowsHealthy := bBrokerHealthy;
END_IF

(* Rising edge of the MQTT session, which is what the birth message wants - not
   bBrokerHealthy, because announcing availability is about having a session to
   announce it on. *)
fbMQTTConnectTrigger(CLK := stMQTTInfo.MQTT_CONNECTED);

(* allow the pulse generator to generate a pulse, used for birth message hartbeat *)
fbMQTTBirthHartbeat(ENQ:=TRUE, PTH:=T#0S, PTL:=GVL_MQTT.MQTTAvailabilityHartbeatTime);

(* Check if this is a new connection due to startup or connection issues *)
IF initMqtt AND (fbMQTTConnectTrigger.Q OR fbMQTTBirthHartbeat.Q) THEN
	bMQTTPublishBirth := TRUE;
END_IF

(* On connect or reconnect publish a birth message using the dedicated birth publisher *)
(* Gated on SendDone: handing the birth publisher a new message while its
   previous publish is still outstanding is the same fault the pool workers
   had, and the flag stays set so the birth goes out as soon as it is free. *)
IF bMQTTPublishBirth AND fbMQTTBirthPublisher.SendDone THEN
	fbMQTTBirthPublisher.PublishMessage(MqttMessage := stMQTTBirthMessage);
	bMQTTPublishBirth:=FALSE;
END_IF


(* Check if Mqtt is initialized AND if there are elements on the queue to process AND if a stMQTTBirthMessage has been published successfully *)
IF initMqtt AND GVL_MQTT.fbMqttPublishQueue.HasMessage() AND bMQTTPublishBirth = FALSE AND fbMQTTBirthPublisher.SendDone THEN	
	(* Loop through all free afbPublishers untill there are no more elements in the queue or no more free afbPublishers *)
	FOR udiI:=0 TO (cudiPublishers-1) DO			
		(* use the afbPublishers that are free  *)
		IF afbPublishers[udiI].SendDone AND GVL_MQTT.fbMqttPublishQueue.HasMessage() THEN	
			(* Pass message from the queue to a publisher *)
			afbPublishers[udiI].PublishMessage(MqttMessage:= GVL_MQTT.fbMqttPublishQueue.GetMessage());
		ELSIF NOT GVL_MQTT.fbMqttPublishQueue.HasMessage() THEN
			(* Queue is empty, jump out of the for loop	*)
			EXIT;	
		END_IF
	END_FOR
END_IF


(* If MQTT is initialized, let the MqttPublishWorkers do their work *)
IF initMqtt THEN	
	MQTT_IN_OUT.clientFB(
		MQTT_IN_OUT:= MQTT_IN_OUT, 
		ENABLE:= bMqttEnable, 
		URL:= GVL_MQTT.broker, 
		TIMEOUT:= T#1S, 
		TLS:= FALSE);		
		
	fbMQTTBirthPublisher();
	
	FOR udiI := 0 TO (cudiPublishers-1) DO
  		afbPublishers[udiI]();
	END_FOR

END_IF

(* --- Reconnect supervision -------------------------------------------------
   Every reconnect attempt costs one 'offline' on the availability topic, so the
   rate of attempts is the rate of the will. MqttClient never leaves politely on
   a fault - step 40 sets COM.MQTT_ABORT, which closes the socket without a
   DISCONNECT packet - and it has no idea whether trying again is working, so
   left alone it will hammer a broker for as long as the fault lasts.

   Two things happen here. The pause between attempts doubles while attempts
   keep failing, so a fault costs a message a minute rather than three a second;
   and a client that has achieved nothing for a long time is switched off for a
   while, which is both quieter and the only graceful exit available - ENABLE
   going FALSE takes the client through step 50, where COM.MQTT_ABORT stays
   clear and MQTT_CONTROL sends a real DISCONNECT, so the broker has no will to
   fire at all. *)
fbSessionStable(IN := stMQTTInfo.MQTT_CONNECTED, PT := GVL_MQTT.tMqttSessionStable);
fbSessionDrop(CLK := stMQTTInfo.MQTT_CONNECTED);

IF fbSessionDrop.Q THEN
	udiSessionDrops := udiSessionDrops + 1;
	udiSessionDropsTotal := udiSessionDropsTotal + 1;
	(* Doubling by addition: TIME + TIME is defined, where multiplying a TIME by
	   a literal invites an implicit conversion nobody wants to read. *)
	IF tMqttRest < GVL_MQTT.tMqttReconnectRestMax THEN
		tMqttRest := tMqttRest + tMqttRest;
	END_IF
	IF tMqttRest > GVL_MQTT.tMqttReconnectRestMax THEN
		tMqttRest := GVL_MQTT.tMqttReconnectRestMax;
	END_IF
END_IF

IF fbSessionStable.Q THEN
	(* A session this old is a working one, so forget the backoff. Report what it
	   took to get here as well: a storm that has ended leaves no other trace,
	   and the count is the difference between a flapping link and a clean
	   restart. *)
	IF NOT bSessionWasStable THEN
		bSessionWasStable := TRUE;
		IF udiSessionDrops > 0 THEN
			GVL_MQTT.PLC_Device.SendLogMessage(CONCAT('MQTT session stable after ',
				CONCAT(UDINT_TO_STRING(udiSessionDrops), ' dropped sessions')));
		END_IF
		udiSessionDrops := 0;
	END_IF
	tMqttRest := GVL_MQTT.tMqttReconnectRestMin;
ELSIF NOT stMQTTInfo.MQTT_CONNECTED THEN
	bSessionWasStable := FALSE;
END_IF

(* The client reads this in step 70, which it reaches between every attempt once
   MQTT_INIT has set RestAfterDisconect. Writing it every cycle rather than on
   the edge keeps one owner for the value. *)
MQTT_IN_OUT.RestTime := tMqttRest;

(* A stall is a client that has not held a working session for a long time. It
   is not going to fix itself by trying again sooner, so it stops trying for a
   while. The count is kept because it is the one symptom that says the fault is
   here rather than at the broker. *)
fbMqttStalled(IN := bMqttEnable AND NOT fbSessionStable.Q, PT := GVL_MQTT.tMqttStall);
fbMqttCoolDown(IN := NOT bMqttEnable, PT := GVL_MQTT.tMqttStallCoolDown);

IF fbMqttStalled.Q THEN
	bMqttEnable := FALSE;
	udiMqttCoolDowns := udiMqttCoolDowns + 1;
END_IF
IF fbMqttCoolDown.Q THEN
	bMqttEnable := TRUE;
END_IF

                      
END_ACTION

ACTION MQTT_INIT:
                        
IF NOT initMqtt THEN
	initMqtt := TRUE;
	(* Basic MQTT config *)
	MQTT_IN_OUT.ClientID := GVL_MQTT.clientID;
	
	(* Set the LWT topic / payload *)
	MQTT_IN_OUT.BuildWillTopicAndMessage := FALSE;
	MQTT_IN_OUT.WillTopicBase := '';
	MQTT_IN_OUT.ClientWillTopic := GVL_MQTT.MqttAvailabilityTopic;
	MQTT_IN_OUT.ClientWillMessage := GVL_MQTT.MqttAvailabilityOfflinePayload;
	
	(* Rest between reconnect attempts instead of going straight round again.
	   The library only honours RestTime when this is set: with it FALSE, step 60
	   returns to step 0 on the next cycle and the retry rate is whatever the task
	   allows. MQTT_PUBLISH owns the value in RestTime and moves it as the
	   connection behaves. *)
	MQTT_IN_OUT.RestAfterDisconect := TRUE;
	MQTT_IN_OUT.RestTime := tMqttRest;
	
	(* Set the birth message *)
	stMQTTBirthMessage.Payload := GVL_MQTT.MqttAvailabilityOnlinePayload;
	stMQTTBirthMessage.Topic := GVL_MQTT.MqttAvailabilityTopic;
	stMQTTBirthMessage.Qos := GVL_MQTT.MQTT_QOS_EXACTLY_ONCE;
	stMQTTBirthMessage.MqttRetain := FALSE;
	
	(* Nothing is connected yet, so start U1 from the disconnected state and record
	   that that is what it shows. Without this the LED keeps whatever the runtime
	   left on it, because MQTT_PUBLISH only writes on a change and at a cold start
	   its remembered state and the real state already agree. *)
	PFC.SetLed(which := PFC.LED.U1, how := PFC.LedState.BLINK_RED);
	bLedShowsHealthy := FALSE;
	
	(* Configure the dedicated MQTTBirth publisher *)
	fbMQTTBirthPublisher.Init(inputMQTT_IN_OUT:= ADR(MQTT_IN_OUT));
	
	(* Configure the pulse generator for the birth message hartbeat *)
	 fbMQTTBirthHartbeat(ENQ:=TRUE, PTH:=T#0S, PTL:=GVL_MQTT.MQTTAvailabilityHartbeatTime);
	
	(* INIT MQTT PUBLISH STUFF *)
	FOR udiIcounter := 0 TO (cudiPublishers-1) DO		
		afbPublishers[udiIcounter].Init(inputMQTT_IN_OUT:= ADR(MQTT_IN_OUT));
	END_FOR 
	
	(* INIT MQTT SUBSCRIBE STUFF *)
	fbSubscriberFbOutputSwitchMqtt.SetMqttInOut(MQTT_IN_OUT:= MQTT_IN_OUT);	
	fbSubscriberFbOutputCoverMqtt.SetMqttInOut(MQTT_IN_OUT:= MQTT_IN_OUT);
	fbSubscriberFbDimmerMqtt.SetMqttInOut(MQTT_IN_OUT:= MQTT_IN_OUT);
	fbSubscriberFbRs485Mqtt.SetMqttInOut(MQTT_IN_OUT:= MQTT_IN_OUT);
	fbSubscriberFbHvacMqtt.SetMqttInOut(MQTT_IN_OUT:= MQTT_IN_OUT);
END_IF


                      
END_ACTION

ACTION MQTT_SUBSCRIBE:
                        (* If MQTT is initialized, let the subscriber(s) do its work *)
IF initMqtt THEN
	
	(* The clientFB call deliberately lives only in MQTT_PUBLISH. Both actions run
	   every scan, so calling it here as well advanced one client instance's state
	   machine twice per cycle in a freewheeling task. *)

	fbSubscriberFbOutputSwitchMqtt(
		Subscribe:= TRUE, 
		Topic:= ADR(GVL_MQTT.MqttSubSwitchTopic), 
		QoSSubscribe:= GVL_MQTT.MQTT_QOS_EXACTLY_ONCE, 
		ExpectingString:= TRUE, 
		Callback:= GVL_MQTT.collector_FB_OUTPUT_SWITCH_MQTT,
	);	
	fbSubscriberFbOutputCoverMqtt(
		Subscribe:= TRUE, 
		Topic:= ADR(GVL_MQTT.MqttSubCoverTopic), 
		QoSSubscribe:= GVL_MQTT.MQTT_QOS_EXACTLY_ONCE, 
		ExpectingString:= TRUE, 
		Callback:= GVL_MQTT.collector_FB_OUTPUT_COVER_MQTT,
	);	
	fbSubscriberFbDimmerMqtt(
		Subscribe:= TRUE, 
		Topic:= ADR(GVL_MQTT.MqttSubDimmerTopic), 
		QoSSubscribe:= GVL_MQTT.MQTT_QOS_EXACTLY_ONCE, 
		ExpectingString:= TRUE, 
		Callback:= GVL_MQTT.collector_FB_DIMMER_MQTT,
	);
	fbSubscriberFbRs485Mqtt(
		Subscribe:= TRUE, 
		Topic:= ADR(GVL_MQTT.MqttSubRS485Topic), 
		QoSSubscribe:= GVL_MQTT.MQTT_QOS_EXACTLY_ONCE,
		ExpectingString:= TRUE, 
		Callback:= GVL_MQTT.collector_FB_RS485_MQTT,
	);
	fbSubscriberFbHvacMqtt(
		Subscribe:= TRUE, 
		Topic:= ADR(GVL_MQTT.MqttSubHVACTopic), 
		QoSSubscribe:= GVL_MQTT.MQTT_QOS_EXACTLY_ONCE,
		ExpectingString:= TRUE, 
		Callback:= GVL_MQTT.collector_FB_HVAC_MQTT,
	);
END_IF
                      
END_ACTION
END_PROGRAM

{attribute 'do_checks_for_implicit_code'}
PROGRAM PRG_HVAC
  VAR
    fbThermostat1 : FB_HVAC_THERMOSTAT_MQTT := (FriendlyName := 'Floorheating');  (* The thermostats, pumps and the burner wire themselves from GVL_MQTT on their first cyclic call, driven by FriendlyName. The positional arguments are each block's own FB_init (setpoint limits, run-on times) and are unchanged. fbPump2Collector is the exception: its discovery config carries eight separate valve names, which a single FriendlyName cannot express, so it keeps both of its explicit calls in HVAC_INIT. Floorheating *)
    fbPump1 : FB_HVAC_PUMP_MQTT := (FriendlyName := 'pump floorheating');  (* These timings protect real hardware: a pump that short-cycles wears out, and a valve needs time to open before there is any point pushing water at it. Do not shorten them here to speed up a test - it does not even work, because changing an FB_init argument from a script updates the declaration text while the compiler keeps reading the old InputAssignments (see CLAUDE.md). Write the members at runtime instead, as the test-plc-logic skill does. *)
    fbThermostat2 : FB_HVAC_THERMOSTAT_MQTT := (FriendlyName := 'Radiator 1');  (* Radiators *)
    fbThermostat3 : FB_HVAC_THERMOSTAT_MQTT := (FriendlyName := 'Radiator 2');
    fbPump2Collector : FB_HVAC_COLLECTOR_MQTT;  (* Valve travel: the pump waits this long after heat is first requested. *)
    asCollectorValveNames : ARRAY[1..8] OF STRING(100);  (* Valve names for the collector's discovery config, indexed the same way as its THERMOSTAT and VALVE arrays. Only the wired circuits are named; the rest stay empty and announce no Home Assistant entity. The bound must match VALVE_COUNT in FB_HVAC_COLLECTOR_MQTT, which is the block's own declaration of how many circuits the manifold has. *)
    fbPump2 : FB_HVAC_PUMP_MQTT := (FriendlyName := 'pump collector');
    fbBurnerGas : FB_HVAC_BURNER_MQTT := (FriendlyName := 'gas boiler');  (* Gas boiler *)
    bInitHvacDone : BOOL := FALSE;
  END_VAR

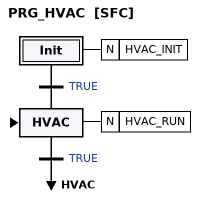
INITIAL_STEP Init:
  HVAC_INIT(N);
END_STEP
TRANSITION FROM Init TO HVAC
  := TRUE;
END_TRANSITION
STEP HVAC:
  HVAC_RUN(N);
END_STEP
TRANSITION FROM HVAC TO HVAC
  := TRUE;
END_TRANSITION

ACTION HVAC_INIT:
                        (* The thermostats, the pumps and the burner now wire and announce themselves from
   their FriendlyName, set where they are declared. What is left here is the one
   block a name cannot describe.

   fbPump2Collector keeps BOTH of its calls, and they belong together: its
   discovery config carries eight separate valve names, so it cannot be driven from
   a single FriendlyName - and because InitMqttDiscovery does nothing until
   InitMqttDone is TRUE, moving only its wiring into the block would leave this
   discovery call running a cycle too early, silently announcing nothing. *)

IF NOT bInitHvacDone THEN
	bInitHvacDone := TRUE;

	fbPump2Collector.InitMqtt(ADR(GVL_MQTT.MqttPubHVACPrefix), ADR(GVL_MQTT.fbMqttPublishQueue));
	asCollectorValveNames[1] := 'Radiator 1';
	asCollectorValveNames[2] := 'Radiator 2';
	fbPump2Collector.InitMqttDiscovery(ADR(GVL_MQTT.PLC_Device), asCollectorValveNames);
END_IF

                      
END_ACTION

ACTION HVAC_RUN:
                        // HVAC flow 1
// 1. A thermostat requests heat once:
// 		1.1 The measured temperature is below the target temperature (hysteresis possible)
//		1.2 The thermostat is in 'heat' mode (or auto mode)
//		1.3 The temperature sensor used in the thermostat is not in error
//		1.4 The measured temperature is not above the configured max temperature
// 2. The Thermostat connects to a heating Valve turning it on/open when heat is required
//		2.1 The heating valve takes X amount of time to switch fully open
//		2.2 The heating valve can only turn on the pump once it's fully open
// 		2.3 The heating valve can only start closing once the pump has completed its minimum cycle time
// 3. The Heating valve is part of PUMP circuit together with other valves:
//		3.1 The pump can only turn off if it has ran for its minimum cycle time
//		3.2 Whenever the pump is running it should request heat from the heating system
// 4. The heating system should provide heat from the moment one pump requires it
//		4.1 A system might have multiple pumps
//		4.2 The heating system might have a minimum cycle time 

// 1. A thermostat requests heat once:
// 		1.1 The measured temperature is below the target temperature (hysteresis possible)
//		1.2 The thermostat is in 'heat' mode (or auto mode)
//		1.3 The temperature sensor used in the thermostat is not in error
//		1.4 The measured temperature is not above the configured max temperature
// 2. The Thermostat connects to a pump turning it on when heat is required
//		2.1 The pump can only turn off if it has ran for its minimum cycle time
//		2.2 Whenever the pump is running it should request heat from the heating system
// 3. The heating system should provide heat from the moment one pump requires it
//		3.1 A system might have multiple pumps
//		3.2 The heating system might have a minimum cycle time 


// FLoorheating
fbThermostat1(MEASURED_TEMP := GVL_RS485.FB_RS485_1WIRE_MULTISENSOR_01.TEMPERATURE, MEASURED_HUM := GVL_RS485.FB_RS485_1WIRE_MULTISENSOR_01.HUMIDITY, SENSOR_VALID := GVL_RS485.FB_RS485_1WIRE_MULTISENSOR_01.DataAvailable AND NOT GVL_RS485.FB_RS485_1WIRE_MULTISENSOR_01.Error);
fbPump1(
	IN := fbThermostat1.OUT
	(* Coil dropped: DO_005..DO_008 are the bench's spare LEDs now, and the
	   cover block uses two of them. The pump logic and its MQTT entity are
	   untouched - only the physical output is gone. *)
);


// Radiators
fbThermostat2(MEASURED_TEMP := GVL_RS485.FB_RS485_1WIRE_MULTISENSOR_01.TEMPERATURE, MEASURED_HUM := GVL_RS485.FB_RS485_1WIRE_MULTISENSOR_01.HUMIDITY, SENSOR_VALID := GVL_RS485.FB_RS485_1WIRE_MULTISENSOR_01.DataAvailable AND NOT GVL_RS485.FB_RS485_1WIRE_MULTISENSOR_01.Error);
fbThermostat3(MEASURED_TEMP := GVL_RS485.FB_RS485_1WIRE_MULTISENSOR_01.TEMPERATURE, MEASURED_HUM := GVL_RS485.FB_RS485_1WIRE_MULTISENSOR_01.HUMIDITY, SENSOR_VALID := GVL_RS485.FB_RS485_1WIRE_MULTISENSOR_01.DataAvailable AND NOT GVL_RS485.FB_RS485_1WIRE_MULTISENSOR_01.Error);

(* Circuit 1 is Radiator 1, circuit 2 is Radiator 2; circuits 3..8 are unwired and
   their valves stay closed. The indices match asCollectorValveNames above and the
   VALVE_n names published to MQTT. *)
fbPump2Collector.THERMOSTAT[1] := fbThermostat2.OUT;
fbPump2Collector.THERMOSTAT[2] := fbThermostat3.OUT;

(* Requirement 2.3 above: the manifold may not start closing while the pump is
   still running out its minimum on-time, or the pump ends up turning against
   shut valves. fbPump2 already computed the signal for it and nothing read it.

   The collector is called before the pump, so it acts on last cycle's value -
   one task cycle of lag on a two-minute timer, and the safe direction: the hold
   is released a cycle late, never engaged a cycle late. *)
fbPump2Collector.PUMP_MIN_ONTIME_ACTIVE := fbPump2.MIN_ONTIME_ACTIVE;

fbPump2Collector();


fbPump2(
	IN := fbPump2Collector.PUMP
);

// Heat source for both pumps
fbBurnerGas(
	IN := fbPump2.HEAT_REQUEST OR fbPump1.HEAT_REQUEST,
	//OUT => DO_013
);
                      
END_ACTION
END_PROGRAM

{attribute 'do_checks_for_implicit_code'}
PROGRAM PRG_RS485
  VAR CONSTANT
    cudiBusBaudrate : UDINT := 9600;  (* What this bus runs at. One rate for the whole pair, so it is written down once: the transport opens the port at it, and commissioning tells a device that disagrees which rate to move to. *)
  END_VAR
  VAR
    InitRS485 : BOOL := FALSE;
    fbRs485Transport : FB_RS485_TRANSPORT_RTU;  (* The wire, and the thing that shares it out. Both are ordinary function blocks now. The Modbus RTU state machine used to live in the RS485_RUN action - about ninety lines of framing, CRC and serial handling inside a program action, where it could not be tested, documented or swapped independently of the program that hosted it. The e!COCKPIT variant that used to sit here commented out is gone rather than lost: WagoAppPlcModbus.FbMbMasterSerial belongs behind the same fbRs485Transport interface as this one, as a second implementation, and so does ModbusFB.ClientSerial. None of them is the program's business. *)
    fbRS485BusController : FB_RS485_BUSCONTROLLER;
    fbRS485Commissioner : FB_RS485_COMMISSIONER;  (* Devices that cannot be spoken to until something has been written into them - one shipping at a baud rate this bus does not use, say. The same argument as the transport above, and it took a second reading of this program to notice: the sweep used to live in RS485_RUN as two hundred lines that named one sensor, its slave address and its registers. A program that owns the bus should not know what is on it. It asks each registered device instead - I_RS485_DEVICE.GetCommissioning - and the device answers with what to probe and what to write. *)
    fbDiagTimer : TON;  (* Thirty-second heartbeat for the bus health topic. The transport's counters are the only instrument this bus has; publishing them beats reading them over an online session that this runtime keeps dropping. *)
    sDiagReport : STRING(400);
  END_VAR

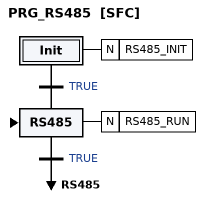
INITIAL_STEP Init:
  RS485_INIT(N);
END_STEP
TRANSITION FROM Init TO RS485
  := TRUE;
END_TRANSITION
STEP RS485:
  RS485_RUN(N);
END_STEP
TRANSITION FROM RS485 TO RS485
  := TRUE;
END_TRANSITION

ACTION RS485_INIT:
                        IF NOT InitRS485 THEN
	InitRS485 := TRUE;

(* THE WIRE.
   COM1 is the only port the PFC200 runtime exposes - COM2, COM3 and COM4 were
   all tried and none of them opens. The port must also have been put into RS485
   mode once per controller with `serialmode RS485` from the CODESYS PLC shell.
   That is a commissioning step: no IEC code can do it, it survives a reboot,
   and until it is done the bus is silent with no error to show for it. *)
fbRs485Transport.Init(
	Port			:= SysCom.SYS_COM_PORTS.SYS_COMPORT1,
	Baudrate		:= cudiBusBaudrate,
	Parity			:= SysCom.SYS_COM_PARITY.SYS_NOPARITY,
	StopBits		:= SysCom.SYS_COM_STOPBITS.SYS_ONESTOPBIT,
	ReplyTimeout	:= T#1S,			(* nothing at all by now means no reply *)
	GapTime			:= T#50MS			(* quiet line ends a frame *)
);

(* WHO GETS IT.
   Registration order no longer decides who is served first: selection resumes
   at a cursor and wraps, so the device registered last is polled as often as
   the device registered first. *)
fbRS485BusController.Init(
	Transport		:= fbRs485Transport,
	StartupDelay	:= T#5S,			(* let the slaves finish booting *)
	SilenceTime		:= T#50MS,			(* between frames, and between transactions *)
	StepTimeout		:= T#3S				(* watchdog on the transport, not on the slave *)
);

fbRS485BusController.RegisterDevice(device := GVL_RS485.FB_RS485_EASTRON_SDM220_1);
fbRS485BusController.RegisterDevice(device := GVL_RS485.FB_RS485_EASTRON_SDM630_1);
//fbRS485BusController.RegisterDevice(device := GVL_RS485.FB_RS485_DUCO_DUCOBOX_HOME);
//fbRS485BusController.RegisterDevice(device := GVL_RS485.FB_RS485_1WIRE_MULTISENSOR_01);
fbRS485BusController.RegisterDevice(device := GVL_RS485.FB_RS485_EASTRON_SDM_POWER_1);
fbRS485BusController.RegisterDevice(device := GVL_RS485.FB_RS485_SEN0492_1);

(* WHAT CANNOT BE SPOKEN TO YET.
   Asked of every device registered above, before the bus controller is allowed to
   start. Nothing here names a device or a register: what has to be written, and
   where, is each device's own answer - see I_RS485_DEVICE.GetCommissioning. A device
   that needs nothing costs one method call.

   It holds the bus off while it runs, because a device being hunted for at some
   other baud rate makes the whole pair unusable for as long as that takes. *)
fbRS485Commissioner.Init(
	Transport			:= fbRs485Transport,
	pController			:= ADR(fbRS485BusController),
	BusBaudrate			:= cudiBusBaudrate,
	pMqttPublishQueue	:= ADR(GVL_MQTT.fbMqttPublishQueue),
	MqttPublishPrefix	:= ADR(GVL_MQTT.MqttPubRS485Prefix),
	Enable				:= GVL_RS485.RS485_COMMISSION_ON_BOOT
);

(* INIT RS485 DEVICE STUFF.
   Nothing to do for the three Eastron meters. Modbus address, poll rate and -
   for the SDM_POWER block - the meter model all reach them through FB_init at
   their declaration in GVL_RS485, and FriendlyName wires up MQTT and Home
   Assistant on the first cyclic call. Registration above is the whole of it. *)

GVL_RS485.FB_RS485_DUCO_DUCOBOX_HOME.InitRS485(
	DataPollingInterval := T#3S,		(* Polling interval for data array *)
	DeviceAddress := 3					(* Device address of the modbus device *)
);

(* Nodes on the bench Ducobox. The names are what Home Assistant shows; the
   topic keeps using the node number, so renaming a room moves no topic.

   What each node IS - valve, sensor, wall control - is not declared here. The
   block reads module type from read parameter 0 and announces the entity set
   that type actually has, so swapping a valve for a sensor needs no edit. *)
GVL_RS485.FB_RS485_DUCO_DUCOBOX_HOME.AddNode(
	FriendlyName := 'Bench node A',
	DataPollingInterval := T#15S
);
GVL_RS485.FB_RS485_DUCO_DUCOBOX_HOME.AddNode(
	FriendlyName := 'Bench node B',
	DataPollingInterval := T#15S
);

GVL_RS485.FB_RS485_DUCO_DUCOBOX_HOME.InitMqtt(
	MQTTPublishPrefix:= ADR(GVL_MQTT.MqttPubRS485Prefix),
	MQTTSubscribePrefix:= ADR(GVL_MQTT.MqttSubRS485Prefix),
	pMqttPublishQueue := ADR(GVL_MQTT.fbMqttPublishQueue),
	pMqttCallbackCollector := ADR(GVL_MQTT.collector_FB_RS485_MQTT)
);

(* Announces the box, and then each component as the bus reports what it is.
   The entity set per component comes from its module type, so nothing here has
   to describe what is on the network. *)
GVL_RS485.FB_RS485_DUCO_DUCOBOX_HOME.InitMqttDiscovery(
	DeviceName := 'Bench Ducobox',
	overruleId := '');


GVL_RS485.FB_RS485_1WIRE_MULTISENSOR_01.InitMqtt(
	MQTTPublishPrefix:= ADR(GVL_MQTT.MqttPubRS485Prefix),
	pMqttPublishQueue := ADR(GVL_MQTT.fbMqttPublishQueue)
);
GVL_RS485.FB_RS485_1WIRE_MULTISENSOR_01.InitMqttDiscovery(
	Device := ADR(GVL_MQTT.OWD_MULTISENSOR_01),
	ParentDevice:= ADR(GVL_MQTT.PLC_Device),
	DeviceName := 'Lab PLC 1-Wire sensorhub',
	SupportsTemperature := TRUE,
	SupportsHumidity := TRUE,
	SupportsDewPoint := TRUE,
	SupportsOwdVoltage := TRUE);


END_IF

                      
END_ACTION

ACTION RS485_RUN:
                        (* Commissioning owns the bus while it runs, so the scheduler is held off until it
   is finished - a device being hunted for at another baud rate makes the pair
   unusable for anything else. With nothing to commission it finishes on its first
   cycle, and this costs one comparison from then on.

   Neither call knows what is on the bus: the commissioner asks every registered
   device whether it needs anything (I_RS485_DEVICE.GetCommissioning), and the bus
   controller asks every registered device whether it wants the bus (HasWork). *)
IF NOT fbRS485Commissioner.Done THEN
	fbRS485Commissioner();
ELSE
	(* The bus controller drives the transport - it calls Service every cycle, which
	   is what opens and re-opens the serial port as well as carrying frames - so
	   there is nothing to do here but call it. *)
	fbRS485BusController();
END_IF

(* --- bus health, published where it can actually be read -----------------------
   The transport's counters are the only instrument this bus has, and reading
   them has meant an online debug session - the least reliable thing in the
   chain on this hardware. Published every thirty seconds instead, retained, so
   the answer to "is the bus healthy" is a topic rather than an expedition.

   The pair that matters is CrcFail against NoReply. Bytes that arrive and never
   frame are a different fault from no bytes at all: the first is framing or
   noise, the second is a device that did not answer. Everything else here is
   context for those two. *)
fbDiagTimer(IN := NOT fbDiagTimer.Q, PT := T#30S);
IF fbDiagTimer.Q THEN
	sDiagReport := CONCAT('ok=', UDINT_TO_STRING(fbRs485Transport.Ok));
	sDiagReport := CONCAT(sDiagReport, ' noreply=');
	sDiagReport := CONCAT(sDiagReport, UDINT_TO_STRING(fbRs485Transport.NoReply));
	sDiagReport := CONCAT(sDiagReport, ' crc=');
	sDiagReport := CONCAT(sDiagReport, UDINT_TO_STRING(fbRs485Transport.CrcFail));
	sDiagReport := CONCAT(sDiagReport, ' short=');
	sDiagReport := CONCAT(sDiagReport, UDINT_TO_STRING(fbRs485Transport.ShortFrame));
	sDiagReport := CONCAT(sDiagReport, ' badaddr=');
	sDiagReport := CONCAT(sDiagReport, UDINT_TO_STRING(fbRs485Transport.BadAddress));
	sDiagReport := CONCAT(sDiagReport, ' badfunc=');
	sDiagReport := CONCAT(sDiagReport, UDINT_TO_STRING(fbRs485Transport.BadFunction));
	sDiagReport := CONCAT(sDiagReport, ' exc=');
	sDiagReport := CONCAT(sDiagReport, UDINT_TO_STRING(fbRs485Transport.Exceptions));
	sDiagReport := CONCAT(sDiagReport, ' lead=');
	sDiagReport := CONCAT(sDiagReport, UDINT_TO_STRING(fbRs485Transport.LeadNulls));
	sDiagReport := CONCAT(sDiagReport, ' trail=');
	sDiagReport := CONCAT(sDiagReport, UDINT_TO_STRING(fbRs485Transport.TrailNulls));
	sDiagReport := CONCAT(sDiagReport, ' tx=');
	sDiagReport := CONCAT(sDiagReport, UDINT_TO_STRING(fbRS485BusController.Transactions));
	sDiagReport := CONCAT(sDiagReport, ' steps=');
	sDiagReport := CONCAT(sDiagReport, UDINT_TO_STRING(fbRS485BusController.StepsExecuted));
	sDiagReport := CONCAT(sDiagReport, ' fail=');
	sDiagReport := CONCAT(sDiagReport, UDINT_TO_STRING(fbRS485BusController.StepFailures));
	sDiagReport := CONCAT(sDiagReport, ' lastfail=dev');
	sDiagReport := CONCAT(sDiagReport, BYTE_TO_STRING(fbRs485Transport.LastFailAddr));
	sDiagReport := CONCAT(sDiagReport, '/fc');
	sDiagReport := CONCAT(sDiagReport, BYTE_TO_STRING(fbRs485Transport.LastFailFunc));
	sDiagReport := CONCAT(sDiagReport, '/n');
	sDiagReport := CONCAT(sDiagReport, UDINT_TO_STRING(fbRs485Transport.LastFailLen));
	(* Messages the publish queue threw away because a lane was full. Silent
   until now, and the one number that says whether MQTT is keeping up. *)
sDiagReport := CONCAT(sDiagReport, ' drop=');
sDiagReport := CONCAT(sDiagReport, UDINT_TO_STRING(GVL_MQTT.fbMqttPublishQueue.DroppedCount));
sDiagReport := CONCAT(sDiagReport, ' [');
	sDiagReport := CONCAT(sDiagReport, fbRs485Transport.LastFailBytes);
	sDiagReport := CONCAT(sDiagReport, ']');

	GVL_MQTT.fbMqttPublishQueue.AddMessageOn(Lane := GVL_MQTT.MQTT_LANE_RS485,
		Payload := sDiagReport,
		Topic := CONCAT(GVL_MQTT.MqttPubRS485Prefix, 'BUS_COUNTERS'),
		Qos := MQTT.QoS.ExactlyOnce,
		MqttRetain := TRUE);
END_IF

(* RS485 devices. Called even while commissioning runs: their bodies only
   publish and self-wire, and the scheduler is the only thing that talks to the
   bus on their behalf. *)
GVL_RS485.FB_RS485_EASTRON_SDM220_1();
GVL_RS485.FB_RS485_DUCO_DUCOBOX_HOME();
GVL_RS485.FB_RS485_1WIRE_MULTISENSOR_01();
GVL_RS485.FB_RS485_EASTRON_SDM630_1();
GVL_RS485.FB_RS485_EASTRON_SDM_POWER_1();
GVL_RS485.FB_RS485_SEN0492_1();

                      
END_ACTION
END_PROGRAM

